FUNCTION_BLOCK "GCS7_E_MYFC_MOZF"	// FB 34
TITLE = MYFC/MOZF Liquids Flow Control
//  
//COPYRIGHT:    (C) 2002  BUHLER AG, CH-9240 UZWIL, SWITZERLAND
//
//PRODUCT:      GCS7
//
//TITLE:        Element MYFC/MOZF Liquids Flow Control
//
//-------------------------------------------------------------------------
//
//IDENT:        AUTHOR:             DEPT:                      DATE:
//
//FB34.3.1      A.Egli              CT3                        01-Dec-2005
//              Parameter Upload Change DBD86-->DBD88
//FB34.3.0      A.Egli              CT3                        05-Jan-2005
//              Parameter Upload (uses DB10)
//FB34.2.3      S.Cable             CDDP                       22-Mar-2004
//              Replace T D [AR1,xxx] with T LD [AR1,xxx]
//              If in Local, but released locally, do not alarm
//FB34.2.2      K.Tischer           CT3                        14-Jan-2004
//              Handling von InManual 
//FB34.2.1      A.Egli              CT3                        22-Dec-2003
//              StCode=6 also when StWaiting                
//FB34.2.0      A.Egli              CT3                        11-Dec-2003
//              InRestdischarge, StCode=6=Emptying 16=Emptying.Warning
//FB34.1.1      A.Egli              CT3                        17-Nov-2003
//              Alarm 90: Fault not DPRemoteControl
//FB34.1.0      A. Egli             CT3                        02-Jun-2002
//              1st Release in S7
//
//-------------------------------------------------------------------------
//
//PURPOSE:      MANUAL : see [MYFCxxMAN]
//
//RESTRICTIONS: S7
//-------------------------------------------------------------------------
//
//=======================================================
//Log Message: 
//------------------------------------------------------
//0     = Fault Cannceled
//1..79 = AlarmLC : Alarmnumber see manual of MYFC
//90   = Remote Control
//91   = StStopped
//92   = StDosing
//93   = StWaiting
//94   = Timeout starting
//95   = Timeout stopping
//96   = Communication fault
//97   = FaultManualMode
//98   = FaultLocalMode
//
//=======================================================
//StCode:  State               
//------------------------------------------------------
//32  StFault         
// 1  StStoppped      
// 2  StStarting      
// 3  StDosing        
//13  StDosing.Manual  
// 4  StWaiting       
// 7  StStopping      
//41  Stopped.HWStop        = StStopped + InHWStop
//51  Stopped.DPFault       = StStopped + InDPFault
//
AUTHOR : EA
FAMILY : GCS7LL
NAME : MYFCMOZE
VERSION : 3.1
VAR
  StCode : INT ;	//Element state code
  InEnable : BOOL ;	//Enable to dosing water
  InLocalWaterControl : BOOL ;	//1=Local Water Control enabled
  InManualWaterControl : BOOL ;	//1=Manual controled water enabled
  InSimulation : BOOL ;	//Simulation with DPSim (only DP)
  InRestdischarge : BOOL ;
  CmdNewJob : BOOL ;	//Clear actual values
  InHWStop : BOOL ;	//No Fault, Element changes to StStopped
  InDPFault : BOOL ;	//No Fault, Element changes to StStopped
  CmdOff : BOOL ;	//Pulse to stopp the element immediately (manual mode)
  CmdOn : BOOL ;	//Pulse to start  the element immediately (manual mode)
  CmdNext : BOOL ;	//Pulse to start the element in automatic mode (see global flags)
  CmdFaultReset : BOOL ;	//Command to reset fault
  InLocal : BOOL ;	//1= Local mode (no fault by start with service switch)
  InManual : BOOL ;	//1=Manual/ 0=Automatic
  InReport : BOOL ;	//Report of all state transitions
  spare37 : BOOL ;
  OutFaultCom : BOOL ;	//Communication fault
  OutFaultMode : BOOL ;	//Wrong mode
  OutFaultRelevant : BOOL ;	//Relevant fault MYFC or MOZF
  spare0403 : BOOL ;
  spare0404 : BOOL ;
  spare0405 : BOOL ;
  OutpEnable : BOOL ;	//24 V Enable signal water dosing
  OutWrongValue : BOOL ;	//Wrong nominal values, rejected by MEAF
  StStopped : BOOL ;	//Element is disabled
  StStarting : BOOL ;	//Element is starting
  StStopping : BOOL ;	//Element is sopping
  StDosing : BOOL ;	//Element is dosing
  StFault : BOOL ;	//Element has a communication or device fault
  StWaiting : BOOL ;	//Element is enabled, Waiting for Product
  OutWarning : BOOL ;	//Warning
  InMoisture : DINT ;	//[0.0 ... 99.9%] or [0..6500.0 l/h]     Is send to LC
  InOffsetMoisture : INT ;	//[-99.99 ... 99.99%]    Is send to MYFC
  InDosingMax : DINT ;	//[0.0 .. 99999.9 l/h] Is send to MYFC
  InProductGroup : INT ;	//[0..99]              Is send to MYFC
  spare18 : DINT ;
  OutMoisture : INT ;	//[0.0 ... 99.9%]      Is read from LC
  OutFlowrateProduct : DINT ;	//[0.. 999999 kg/h]    Is read from MYFC  [de: Istleistung Produkt]
  OutFlowrateWater : DINT ;	//[0.. 6500.0 l/h]    Is read from LC  [de: Istleistung MOZF]
  OutAlarmNrMYFC : INT ;	//Is read from MYFC
  OutAlarmNrMOZF : INT ;	//Is read from LC
  OutTotalProduct : DINT ;	//Is calculated by element
  OutTotalWater : DINT ;	//Is calculated by element
  OutNotErasableWater : DINT ;	//[0..99'999'999.9 l]  Is read from LC
  OutNotErasableProduct : DINT ;	//[0..999'999'999 kg]  Is read from MYFC
  spare52 : DINT ;
  spare56 : INT ;
  OutAlarmNrLog : INT ;
  Par : STRUCT
   ParObjectNo : INT ;	//Is used for communication with PC, e.g. for message
   ParMsgType : INT ;	//Is used for message (translation of state)
   ParHornCode : INT ;	//Is used by horn module
   ParLogOff : BOOL ;	//Report is off
   ParManual : BOOL ;	//Manual mode without interlocking
   ParMOZF : BOOL ;	//1=MOZF / 0=MYFC
   ParDP : BOOL ;	//1=DP / 0=Opto22
   ParFilter : STRUCT
    A05_24VToLow : BOOL ;
    A07ADRange : BOOL ;
    A08ADCalibration : BOOL ;
    A09ADFunction : BOOL ;
    A10ADSupply : BOOL ;
    A11AnalogInput : BOOL ;
    AxxCommunication : BOOL ;	//A12: Serial Interface ; A14=DPFault
    A17InternalCom : BOOL ;
    A26Tolerance : BOOL ;
    A30ZeroTara : BOOL ;
    A38Slide : BOOL ;
    A39Leck : BOOL ;
    A54RelaisMOZF : BOOL ;
    A55Moisture : BOOL ;
    A56TemperatureInternal : BOOL ;
    A57TemperatureExternal : BOOL ;
    A58SignalDumping : BOOL ;
    A59BulkDesity : BOOL ;
    A60Niveau : BOOL ;
    A63LevelProbe : BOOL ;
    A64AlarmMOZE : BOOL ;
    A65MinFlowrate : BOOL ;
    A66MaxFlowrate : BOOL ;
    A67ToleranceWater : BOOL ;
   END_STRUCT ;
   ParComDB : INT ;	//OPTO22: Communication DB
   ParLCIdx : INT ;	//OPTO22: Index of data record
   ParLCAddr : INT ;	//OPTO22: Address of LC Opto22
   ParIOByteNr : INT ;	//PROFIBUS: Address of first input and output byte
   ParMonTime : INT  := 20;	//After this time outputs must be equal inputs
   spare20 : DINT ;
   spare24 : DINT ;
   OutMonTime : INT ;	//Actual time: Monitoring
   OutFlags : STRUCT
    OutFaultResetDone : BOOL ;
    OutAlarmReadAgain : BOOL ;
    OutTestNewAlarm : BOOL ;
    OutRelevantFaultMOZF : BOOL ;	//Relevant fault number
    OutRelevantFaultMYFC : BOOL ;	//Relevant fault number
    OutNoAlarmMOZF : BOOL ;	//Alarmnumber 0 is read form LC
    OutNoAlarmMYFC : BOOL ;	//Alarmnumber 0 is read form LC
    OutComFaultRead : BOOL ;	//Only DP
    OutComFaultSend : BOOL ;	//Only DP
    spare03 : BOOL ;
    spare04 : BOOL ;
    spare05 : BOOL ;
   END_STRUCT ;
   Command : STRUCT 	//Only used with DP Communication
    spare10 : BOOL ;
    spare11 : BOOL ;
    InRestdischarge : BOOL ;
    spare13 : BOOL ;
    spare14 : BOOL ;
    spare15 : BOOL ;
    spare16 : BOOL ;
    AcceptNewDataReady : BOOL ;	//de: Quittierung neue Werte Bereit
    spare2 : BYTE ;
    spare3 : BYTE ;
    CommandReady : BOOL ;	//de: Steuersignale gültig
    spare41 : BOOL ;
    spare42 : BOOL ;
    spare43 : BOOL ;
    spare44 : BOOL ;
    ResetAlarm : BOOL ;	//de: Alarm löschen
    NewSendData : BOOL ;	//de: Aenderung Sendedaten
    AcceptNewRcvData : BOOL ;	//de: Quittierung Aenderung Empfangsdatensatz
   END_STRUCT ;
   Status : STRUCT 	//Only used with DP Communication
    Enable24V : BOOL ;	//Dosing release
    Dosing : BOOL ;	//de: Wasser dosiert
    Remote : BOOL ;	//Remote=1 /Local=0
    Manual : BOOL ;	//de: Hand
    Level : BOOL ;	//1=Covered  de: Sonde Netzgeraet
    Active : BOOL ;	//de: Netzung aktiv
    spare16 : BOOL ;
    NewDataReady : BOOL ;	//de: Neue Werte Bereit
    spare2 : BYTE ;
    spare3 : BYTE ;
    spare40 : BOOL ;
    spare41 : BOOL ;
    spare42 : BOOL ;	//de: Stuerung Remote
    RemoteControlDP : BOOL ;	//de: Sollwertvorgabe Remote
    WrongValue : BOOL ;	//de: Falscher Sollwert
    SumFault : BOOL ;	//de: Sammelalarm
    AcceptNewSendData : BOOL ;	//de: Quittierung Aenderung Sendedaten
    NewRcvData : BOOL ;	//de: Aenderung Empfangsdaten
   END_STRUCT ;
  END_STRUCT ;
END_VAR
VAR_TEMP
  tmpFilter : ARRAY  [0 .. 95 ] OF BOOL ;
  tmpLOGvalue : WORD ;	//LOG value
  tmpCommand : INT ;
  tmpFBNO : INT ;	//Number of the actual FB
  tmpFault : BOOL ;
  tmpOff : BOOL ;
  tmpOn : BOOL ;
  tmpLocal : BOOL ;
  tmpEnable : BOOL ;
  tmpReport : BOOL ;
  tmpLenDyn : DINT ;
  tmpAddr : WORD ;
  tmpReturn : INT ;
  tmpComDB : INT ;
  Set001 : STRUCT
   OutMoistureAc : BYTE ;	//[0.0 ... 99.9%]      Is read from LC
   spare9 : BYTE ;
   OutFlowRateMOZF : INT ;	//[0.. 99999.9 l/h]    Is read from LC  [de: Istleistung MOZF]
   OutFlowRateProduct : DINT ;	//[0.. 999999 kg/h]    Is read from MYFC  [de: Istleistung Produkt]
   OutNotErasableTotalWater : DINT ;	//[0..99'999'999.9 l]  Is read from LC
   spare20 : BYTE ;
   OutRecipeNr : BYTE ;
   OutAlarmNumberMYFC : BYTE ;	//Is read from MYFC
   OutAlarmNumberMOZF : BYTE ;	//Is read from LC
  END_STRUCT ;
  Set136 : STRUCT
   InMoistureNom : INT ;	//[0.00 ... 25.0%]      Is send to LC
   spare10 : INT ;
   InMoistureOffset : INT ;	//[-99.99 ... 99.99%]    Is send to MYFC
   InDosingMax : WORD ;	//[0.0 .. 99999.9 l/h] Is send to MYFC
   InProductGroup : BYTE ;	//[0..99]              Is send to MYFC
   Spare17 : BYTE ;
   Spare18 : DWORD ;
   Spare22 : WORD ;
  END_STRUCT ;
  DPData : STRUCT
   StatusCommand : DWORD ;
   NrSndDataSet : BYTE ;	//de: Nummer Sendedatensatz
   IdxSndDataSet : BYTE ;	//de: Index Sendedatensatz
   NrRcvDataSet : BYTE ;	//de: Nummer Empfangsdatensatz
   IdxRcvDataSet : BYTE ;	//de: Index Empfangsdatensatz
   Data : ARRAY  [1 .. 4 ] OF DINT ;
  END_STRUCT ;
  tmpWtWater : DINT ;
  tmpWtProduct : DINT ;
  tmpCalculate : BOOL ;
  tmpNewAlarmNumber : BOOL ;
  tmpCallBackFuction : BOOL ;	//Call back function is active
  tmpFaultMonitoringStart : BOOL ;
  tmpFaultMonitoringStop : BOOL ;
END_VAR
BEGIN
NETWORK
TITLE =  Start Global
      L     #Par.ParComDB;
      T     #tmpComDB;
      L     34;
      T     #tmpFBNO;
      L     102;
      T     #tmpLenDyn;	//--> Len dynamic data in byte
      SET;
      R     #tmpCalculate;
      R     #tmpCallBackFuction;
      R     #tmpNewAlarmNumber;
      R     #tmpFaultMonitoringStart;
      R     #tmpFaultMonitoringStop;
//tmpLocal
      A     #InLocal;
      AN    #InManual;
      =     #tmpLocal;
NETWORK
TITLE =
      LAR1  P##tmpFilter;
      L     0;
      T     LD [AR1,P#0.0];	//tmpFilter[00..31] [2.3]
      T     LD [AR1,P#0.0];	//tmpFilter[32..63] [2.3]
      T     LD [AR1,P#0.0];	//tmpFilter[64..95] [2.3]
      SET;
      S     #tmpFilter[13];
      S     #tmpFilter[18];
      A     #Par.ParFilter.A05_24VToLow;
      =     #tmpFilter[5];
      A     #Par.ParFilter.A07ADRange;
      =     #tmpFilter[7];
      A     #Par.ParFilter.A08ADCalibration;
      =     #tmpFilter[8];
      A     #Par.ParFilter.A09ADFunction;
      =     #tmpFilter[9];
      A     #Par.ParFilter.A10ADSupply;
      =     #tmpFilter[10];
      A     #Par.ParFilter.A11AnalogInput;
      =     #tmpFilter[11];
      A     #Par.ParFilter.AxxCommunication;
      =     #tmpFilter[12];
      =     #tmpFilter[14];
      A     #Par.ParFilter.A17InternalCom;
      =     #tmpFilter[17];
      A     #Par.ParFilter.A26Tolerance;
      =     #tmpFilter[26];
      A     #Par.ParFilter.A30ZeroTara;
      =     #tmpFilter[30];
      A     #Par.ParFilter.A38Slide;
      =     #tmpFilter[38];
      A     #Par.ParFilter.A39Leck;
      =     #tmpFilter[39];
      A     #Par.ParFilter.A54RelaisMOZF;
      =     #tmpFilter[54];
      A     #Par.ParFilter.A55Moisture;
      =     #tmpFilter[55];
      A     #Par.ParFilter.A56TemperatureInternal;
      =     #tmpFilter[56];
      A     #Par.ParFilter.A57TemperatureExternal;
      =     #tmpFilter[57];
      A     #Par.ParFilter.A58SignalDumping;
      =     #tmpFilter[58];
      A     #Par.ParFilter.A59BulkDesity;
      =     #tmpFilter[59];
      A     #Par.ParFilter.A60Niveau;
      =     #tmpFilter[60];
      A     #Par.ParFilter.A63LevelProbe;
      =     #tmpFilter[63];
      A     #Par.ParFilter.A64AlarmMOZE;
      =     #tmpFilter[64];
      A     #Par.ParFilter.A65MinFlowrate;
      =     #tmpFilter[65];
      A     #Par.ParFilter.A66MaxFlowrate;
      =     #tmpFilter[66];
      A     #Par.ParFilter.A67ToleranceWater;
      =     #tmpFilter[67];
NETWORK
TITLE =  Call back function (***Opto22***)
////*************************************************
////***             O P T O 22                    ***
////*************************************************
//
//This functions are called by FBxxx (COM) 
      A     #Par.ParDP;
      JC    PC;
      OPN   DB [#tmpComDB];
      L     0;
      L     DBW 32;	//COM.Element.CODE;
      ==I;
      JC    PC;
//Check if object has moved
      L     #Par.ParObjectNo;
      L     DBD 60;	//COM.LC0.AddrPara;       
      ==D;
      JC    COok;
      BEC;
//=============================================
COok: S     #tmpCallBackFuction;
      L     DBB 76;	//COM.Telegram.Command;
      T     #tmpCommand;
      L     1;
      L     DBW 32;	//COM.Element.CODE;
      ==I;
      JC    Send;
      L     2;
      ==I;
      JC    Rcv;
      L     4;	//NAK
      L     DBW 32;	//COM.Element.CODE;
      ==I;
      S     #OutFaultCom;	//fault MYEB communication
      BEU;
//--------------------------
//Send C
//--------------------------
Send: NOP   0;
      L     #tmpCommand;
      L     'C';
      <>I;
      JC    SndF;
// command 1
      A     #CmdFaultReset;
      =     #Par.Command.ResetAlarm;
      R     #CmdFaultReset;
// command 1
      L     0;	//Character offset
      T     DBW 40;	//COM.Element.AddrOffset
      L     0;
      T     DBD 36;	//COM.Element.InOutValue
      A     #Par.Command.ResetAlarm;
      =     DBX 39.0;	//-->ResetAlarm
      A     #InRestdischarge;	//                        [2.0]
      =     DBX 39.1;	//-->InRestdischarge      [2.0]
      A     #OutpEnable;
      =     DBX 39.7;	//-->Enable24V for OPTOSIM
      L     32;	//Convert Hex to 2-ASCII
      T     DBW 0;	//COM.CODE
      CDB;	//ComDB->Instanz-DB
      UC    "GCS7_RS485Ctrl";	//Convert (CODE=DBW0)
      CDB;	//ElementDB->Instanz-DB
// InMoistureNom    
      L     2;	//Character offset
      T     DBW 40;	//COM.Element.AddrOffset
      L     #InMoisture;
      T     DBD 36;	//COM.Element.InOutValue
      L     13;	//Convert DInt to 3-ASCII
      T     DBW 0;	//COM.CODE
      CDB;	//ComDB->Instanz-DB
      UC    "GCS7_RS485Ctrl";	//Convert (CODE=DBW0)
      CDB;	//ElementDB->Instanz-DB
// InMoistureOffset    
      L     5;	//Character offset
      T     DBW 40;	//COM.Element.AddrOffset
      L     #InOffsetMoisture;	//[4.0]
      T     DBD 36;	//COM.Element.InOutValue
      L     15;	//Convert DInt to 5-ASCII
      T     DBW 0;	//COM.CODE
      CDB;	//ComDB->Instanz-DB
      UC    "GCS7_RS485Ctrl";	//Convert (CODE=DBW0)
      CDB;	//ElementDB->Instanz-DB
// InDosingMax    
      L     10;	//Character offset
      T     DBW 40;	//COM.Element.AddrOffset
      L     #InDosingMax;	// 
      T     DBD 36;	//COM.Element.InOutValue
      L     16;	//Convert DInt to 6-ASCII
      T     DBW 0;	//COM.CODE
      CDB;	//ComDB->Instanz-DB
      UC    "GCS7_RS485Ctrl";	//Convert (CODE=DBW0)
      CDB;	//ElementDB->Instanz-DB
// InProductGroup    
      L     16;	//Character offset
      T     DBW 40;	//COM.Element.AddrOffset
      L     #InProductGroup;	// 
      T     DBD 36;	//COM.Element.InOutValue
      L     12;	//Convert DInt to 2-ASCII
      T     DBW 0;	//COM.CODE
      CDB;	//ComDB->Instanz-DB
      UC    "GCS7_RS485Ctrl";	//Convert (CODE=DBW0)
      CDB;	//ElementDB->Instanz-DB
// spare    
      L     18;	//Character offset
      T     DBW 40;	//COM.Element.AddrOffset
      L     0;	// 
      T     DBD 36;	//COM.Element.InOutValue
      L     18;	//Convert DInt to 8-ASCII
      T     DBW 0;	//COM.CODE
      CDB;	//ComDB->Instanz-DB
      UC    "GCS7_RS485Ctrl";	//Convert (CODE=DBW0)
      CDB;	//ElementDB->Instanz-DB
// spare    
      L     24;	//Character offset
      T     DBW 40;	//COM.Element.AddrOffset
      L     0;	// 
      T     DBD 36;	//COM.Element.InOutValue
      L     16;	//Convert DInt to 6-ASCII
      T     DBW 0;	//COM.CODE
      CDB;	//ComDB->Instanz-DB
      UC    "GCS7_RS485Ctrl";	//Convert (CODE=DBW0)
      CDB;	//ElementDB->Instanz-DB
      L     30;	//Lenght in byte
      T     DBW 78;	//COM.Telegram.Len
      L     50;	//Lenght in byte
      T     DBW 86;	//COM.Telegram.LenAnswer
      BEU;
//--------------------------
//Send F
//--------------------------
SndF: NOP   0;
      L     #tmpCommand;
      L     'F';
      <>I;
      JC    SndZ;
// command 1
      A     #CmdFaultReset;
      =     #Par.Command.ResetAlarm;
      R     #CmdFaultReset;
// command 1
      L     0;	//Character offset
      T     DBW 40;	//COM.Element.AddrOffset
      L     0;
      T     DBD 36;	//COM.Element.InOutValue
      A     #Par.Command.ResetAlarm;
      =     DBX 39.0;	//-->ResetAlarm
      A     #OutpEnable;
      =     DBX 39.7;	//-->Enable24V for OPTOSIM
      L     32;	//Convert Hex to 2-ASCII
      T     DBW 0;	//COM.CODE
      CDB;	//ComDB->Instanz-DB
      UC    "GCS7_RS485Ctrl";	//Convert (CODE=DBW0)
      CDB;	//ElementDB->Instanz-DB
// InMoistureNom    
      L     2;	//Character offset
      T     DBW 40;	//COM.Element.AddrOffset
      L     #InMoisture;
      T     DBD 36;	//COM.Element.InOutValue
      L     16;	//Convert DInt to 6-ASCII
      T     DBW 0;	//COM.CODE
      CDB;	//ComDB->Instanz-DB
      UC    "GCS7_RS485Ctrl";	//Convert (CODE=DBW0)
      CDB;	//ElementDB->Instanz-DB
// spare    
      L     8;	//Character offset
      T     DBW 40;	//COM.Element.AddrOffset
      L     0;	// 
      T     DBD 36;	//COM.Element.InOutValue
      L     12;	//Convert DInt to 2-ASCII
      T     DBW 0;	//COM.CODE
      CDB;	//ComDB->Instanz-DB
      UC    "GCS7_RS485Ctrl";	//Convert (CODE=DBW0)
      CDB;	//ElementDB->Instanz-DB
      L     10;	//Lenght in byte
      T     DBW 78;	//COM.Telegram.Len
      L     30;	//Lenght in byte
      T     DBW 86;	//COM.Telegram.LenAnswer
SndZ: BEU;
//--- Get done ---------------
//Copy reveived data to element
//--------------------------
//Receive C
//--------------------------
Rcv:  R     #OutFaultCom;
      L     #tmpCommand;
      L     'C';
      <>I;
      JC    RcvF;
      A     #Par.OutFlags.OutFaultResetDone;	//[1.2]
      S     #Par.OutFlags.OutTestNewAlarm;	//[1.2]
      A     #Par.Command.ResetAlarm;	//    [1.2]
      =     #Par.OutFlags.OutFaultResetDone;	// [1.2] 
//LC status
      L     0;	//Character offset
      T     DBW 40;	//COM.Element.AddrOffset
      L     42;	//Convert 2-ASCII to Hex
      T     DBW 0;	//COM.CODE
      CDB;	//ComDB->Instanz-DB
      UC    "GCS7_RS485Ctrl";	//Convert (CODE=DBW0)
      CDB;	//ElementDB->Instanz-DB
      CALL  "SIEMENS_BLKMOV" (
           SRCBLK                   := DBB 39,
           RET_VAL                  := #tmpReturn,
           DSTBLK                   := #Par.Status);
//OutMoistureAc
      L     2;	//Character offset
      T     DBW 40;	//COM.Element.AddrOffset
      L     23;	//Convert 3-ASCII to DInt
      T     DBW 0;	//COM.CODE
      CDB;	//ComDB->Instanz-DB
      UC    "GCS7_RS485Ctrl";	//Convert (CODE=DBW0)
      CDB;	//ElementDB->Instanz-DB
      L     DBD 36;	//COM.Element.InOutValue
      T     #OutMoisture;
//OutFlowRateProduct
      L     5;	//Character offset
      T     DBW 40;	//COM.Element.AddrOffset
      L     26;	//Convert 6-ASCII to DInt
      T     DBW 0;	//COM.CODE
      CDB;	//ComDB->Instanz-DB
      UC    "GCS7_RS485Ctrl";	//Convert (CODE=DBW0)
      CDB;	//ElementDB->Instanz-DB
      L     DBD 36;	//COM.Element.InOutValue
      T     #OutFlowrateProduct;
//OutFlowRateMOZF
      L     11;	//Character offset
      T     DBW 40;	//COM.Element.AddrOffset
      L     26;	//Convert 6-ASCII to DInt
      T     DBW 0;	//COM.CODE
      CDB;	//ComDB->Instanz-DB
      UC    "GCS7_RS485Ctrl";	//Convert (CODE=DBW0)
      CDB;	//ElementDB->Instanz-DB
      L     DBD 36;	//COM.Element.InOutValue
      T     #OutFlowrateWater;
//OutNotErasableTotalWater
      L     17;	//Character offset
      T     DBW 40;	//COM.Element.AddrOffset
      L     29;	//Convert 9-ASCII to DInt
      T     DBW 0;	//COM.CODE
      CDB;	//ComDB->Instanz-DB
      UC    "GCS7_RS485Ctrl";	//Convert (CODE=DBW0)
      CDB;	//ElementDB->Instanz-DB
      L     DBD 36;	//COM.Element.InOutValue
      T     #tmpWtWater;
//OutNotErasableTotalProd
      L     26;	//Character offset
      T     DBW 40;	//COM.Element.AddrOffset
      L     29;	//Convert 9-ASCII to DInt
      T     DBW 0;	//COM.CODE
      CDB;	//ComDB->Instanz-DB
      UC    "GCS7_RS485Ctrl";	//Convert (CODE=DBW0)
      CDB;	//ElementDB->Instanz-DB
      L     DBD 36;	//COM.Element.InOutValue
      T     #tmpWtProduct;
//OutAlarmNumberMYFC
      L     35;	//Character offset
      T     DBW 40;	//COM.Element.AddrOffset
      L     22;	//Convert 2-ASCII to DInt
      T     DBW 0;	//COM.CODE
      CDB;	//ComDB->Instanz-DB
      UC    "GCS7_RS485Ctrl";	//Convert (CODE=DBW0)
      CDB;	//ElementDB->Instanz-DB
      L     DBD 36;	//COM.Element.InOutValue
      T     #Set001.OutAlarmNumberMYFC;
//OutAlarmNumberMOZF
      L     37;	//Character offset
      T     DBW 40;	//COM.Element.AddrOffset
      L     22;	//Convert 2-ASCII to DInt
      T     DBW 0;	//COM.CODE
      CDB;	//ComDB->Instanz-DB
      UC    "GCS7_RS485Ctrl";	//Convert (CODE=DBW0)
      CDB;	//ElementDB->Instanz-DB
      L     DBD 36;	//COM.Element.InOutValue
      T     #Set001.OutAlarmNumberMOZF;
      SET;
      S     #tmpCalculate;
      S     #tmpNewAlarmNumber;
      JU    RCal;	// -->Calculate
//--------------------------
//Receive F
//--------------------------
RcvF: R     #OutFaultCom;
      L     #tmpCommand;
      L     'F';
      <>I;
      BEC;
      A     #Par.OutFlags.OutFaultResetDone;	//[1.2]
      S     #Par.OutFlags.OutTestNewAlarm;	//[1.2]
      A     #Par.Command.ResetAlarm;	//    [1.2]
      R     #CmdFaultReset;
      =     #Par.OutFlags.OutFaultResetDone;	// [1.2] 
//LC status
      L     0;	//Character offset
      T     DBW 40;	//COM.Element.AddrOffset
      L     42;	//Convert 2-ASCII to Hex
      T     DBW 0;	//COM.CODE
      CDB;	//ComDB->Instanz-DB
      UC    "GCS7_RS485Ctrl";	//Convert (CODE=DBW0)
      CDB;	//ElementDB->Instanz-DB
      L     DBD 36;	//COM.Element.InOutValue
      CALL  "SIEMENS_BLKMOV" (
           SRCBLK                   := DBB 39,
           RET_VAL                  := #tmpReturn,
           DSTBLK                   := #Par.Status);
//OutFlowRateMOZF
      L     2;	//Character offset
      T     DBW 40;	//COM.Element.AddrOffset
      L     26;	//Convert 6-ASCII to DInt
      T     DBW 0;	//COM.CODE
      CDB;	//ComDB->Instanz-DB
      UC    "GCS7_RS485Ctrl";	//Convert (CODE=DBW0)
      CDB;	//ElementDB->Instanz-DB
      L     DBD 36;	//COM.Element.InOutValue
      T     #OutFlowrateWater;
//OutNotErasableTotalWater
      L     8;	//Character offset
      T     DBW 40;	//COM.Element.AddrOffset
      L     29;	//Convert 9-ASCII to DInt
      T     DBW 0;	//COM.CODE
      CDB;	//ComDB->Instanz-DB
      UC    "GCS7_RS485Ctrl";	//Convert (CODE=DBW0)
      CDB;	//ElementDB->Instanz-DB
      L     DBD 36;	//COM.Element.InOutValue
      T     #tmpWtWater;
      L     0;
      T     #tmpWtProduct;
//OutAlarmNumberMOZF
      L     17;	//Character offset
      T     DBW 40;	//COM.Element.AddrOffset
      L     22;	//Convert 2-ASCII to DInt
      T     DBW 0;	//COM.CODE
      CDB;	//ComDB->Instanz-DB
      UC    "GCS7_RS485Ctrl";	//Convert (CODE=DBW0)
      CDB;	//ElementDB->Instanz-DB
      L     DBD 36;	//COM.Element.InOutValue
      T     #Set001.OutAlarmNumberMOZF;
      L     0;
      T     #Set001.OutAlarmNumberMYFC;
      SET;
      S     #tmpCalculate;
      S     #tmpNewAlarmNumber;
      JU    RCal;	//-->Calculate Total
NETWORK
TITLE = PC Control
//=== Test Object number =====================
PC:   L     "SYS_DirectCtrlDB".PC.ObjectNo;	//PCControl.ObjectNo
      L     #Par.ParObjectNo;	//Input ObjectNo
      <>I;
      JC    Ctrl;
//=== Test OType      ========================
      L     1034;	//Input object type
      L     "SYS_DirectCtrlDB".PC.ObjectType;	//PCControl.ObjectType
      <>I;
      JC    Ctrl;
//=== Test Handshake =========================
      A     "SYS_DirectCtrlDB".PC.Hsk.FExamine;	//Handshake.FExamine
      JC    pExa;
      A     "SYS_DirectCtrlDB".PC.Hsk.FDefineCmd;	//Handshake.FDefineCmd
      JC    pCmd;
      A     "SYS_DirectCtrlDB".PC.Hsk.FDefinePara;	//Handshake.FDefinePara
      JC    pPar;
pIni: L     2;	//FcInit
      UC    "SYS_DirectCtrl";
      JU    Ctrl;
// Write parameter 
pPar: LAR1  P#DBX 58.0;	//PCControl.Value[1]
      L     #tmpLenDyn;
      SLD   3;
      +AR1;	//PCControl.Value[x]
      L     DBW [AR1,P#20.0];	//PCControl.Value[x+6]
      T     #Par.ParMonTime;
//Write new commands from PC to Interface of group 
pCmd: A     "SYS_DirectCtrlDB".PC.Cmd1[8];	// CmdOff
      AN    "GCS7_Gr_OutManualOff";	//Global.OutManualOff 
      S     #CmdOff;
      A     "SYS_DirectCtrlDB".PC.Cmd1[9];	// CmdOn
      AN    "GCS7_Gr_OutManualOff";	//Global.OutManualOff
      S     #CmdOn;
      A     "SYS_DirectCtrlDB".PC.Cmd1[10];	// CmdNext
      S     #CmdNext;
      A     "SYS_DirectCtrlDB".PC.Cmd1[11];	// CmdFaultReset
      S     #CmdFaultReset;
      A     "SYS_DirectCtrlDB".PC.Cmd1[1];	//Cmd1[1]
      S     #InLocalWaterControl;
      R     #InManualWaterControl;	// CmdManualOn
      A     "SYS_DirectCtrlDB".PC.Cmd1[2];
      S     #InManualWaterControl;	// CmdReportOn
      A     "SYS_DirectCtrlDB".PC.Cmd1[3];
      R     #InLocalWaterControl;	// CmdManualOff
      R     #InManualWaterControl;
      A     "SYS_DirectCtrlDB".PC.Cmd1[5];	//Cmd1[5]  =CmdNewJob
      S     #CmdNewJob;
      A     "SYS_DirectCtrlDB".PC.Cmd1[13];	// CmdManualOn
      S     #InManual;
      A     "SYS_DirectCtrlDB".PC.Cmd1[14];	// CmdReportOn
      S     #InReport;
      A     "SYS_DirectCtrlDB".PC.Cmd2[13];	// CmdManualOff
      R     #InManual;
      A     "SYS_DirectCtrlDB".PC.Cmd2[14];	// CmdReportOff
      R     #InReport;
//Define Value
      AN    "SYS_DirectCtrlDB".PC.Hsk.FDefineValue;	// PC.Hsk.FDefineValue
      ON    #InManual;
      JC    pIni;
      LAR1  P#DBX 58.0;
      L     DBD [AR1,P#6.0];
      T     #InMoisture;
      L     DBW [AR1,P#10.0];
      T     #InOffsetMoisture;
      L     DBD [AR1,P#12.0];
      T     #InDosingMax;
      L     DBW [AR1,P#16.0];
      T     #InProductGroup;
      JU    pIni;
pExa: TAR2;	//Address dynamic datas
      T     "SYS_DirectCtrlDB".GC.InDynAddr;	//-->PCControl.GC.InDynAddr
      L     #tmpLenDyn;	//Length dynamic datas
      T     "SYS_DirectCtrlDB".GC.InDynLen;	//-->PCControl.GC.InDynLen
      L     0;	//Address parameter data
      T     "SYS_DirectCtrlDB".GC.InParaAddr;	//-->PCControl.GC.InParaAddr
      L     0;	//Length parameter
      T     "SYS_DirectCtrlDB".GC.InParaLen;	//-->PCControl.GC.InParaLen
      L     1;	//Code FcExamine
      UC    "SYS_DirectCtrl";
      L     0;	//Revision
      T     "SYS_DirectCtrlDB".GC.Revision;
Ctrl: NOP   0;
NETWORK
TITLE = [3.0] LCParameter
      L     #Par.ParObjectNo;
      L     "SYS_DirectCtrlLCDB".PC.ObjectNo;
      <>I;
      O     #Par.ParDP;
      JC    LCP0;
      T     "SYS_DirectCtrlLCDB".GC.InObjectNo;
      L     #Par.ParComDB;
      T     "SYS_DirectCtrlLCDB".GC.InDBNr;
      L     #Par.ParLCAddr;
      T     "SYS_DirectCtrlLCDB".GC.InLCAddr;
LCP0: NOP   0;
NETWORK
TITLE = Read data from LC (**DP**)
////*************************************************
////***            DP Communication              ***
////*************************************************
//
      AN    #Par.ParDP;
      JC    rcv0;
      L     #Par.ParIOByteNr;
      T     #tmpAddr;
      A     #InSimulation;
      JC    rSim;
      CALL  "SIEMENS_DPRD_DAT" (
           LADDR                    := #tmpAddr,
           RET_VAL                  := #tmpReturn,
           RECORD                   := #DPData);
      L     #tmpReturn;
      L     0;
      <>I;
      =     #Par.OutFlags.OutComFaultRead;
      JC    rcv0;
      JU    rDP;
//read from Simulation
rSim: R     #Par.OutFlags.OutComFaultRead;
      A     "GCS7_Gr_SimDPtoImage";
      L     P#I 0.0;
      JC    rDB1;
      OPN   "TEST_IOSimuliInput";
      L     P#DBX 0.0;
rDB1: L     #Par.ParIOByteNr;
      SLD   3;
      +D;
      LAR1;
      L     D [AR1,P#0.0];
      T     #DPData.StatusCommand;
      L     B [AR1,P#4.0];
      T     #DPData.NrSndDataSet;
      L     B [AR1,P#5.0];
      T     #DPData.IdxSndDataSet;
      L     B [AR1,P#6.0];
      T     #DPData.NrRcvDataSet;
      L     B [AR1,P#7.0];
      T     #DPData.IdxRcvDataSet;
      L     D [AR1,P#8.0];
      T     #DPData.Data[1];
      L     D [AR1,P#12.0];
      T     #DPData.Data[2];
      L     D [AR1,P#16.0];
      T     #DPData.Data[3];
      L     D [AR1,P#20.0];
      T     #DPData.Data[4];
//==Copy Status===============
rDP:  L     #DPData.NrRcvDataSet;
      L     0;
      ==I;
      JC    R001;
      CALL  "SIEMENS_BLKMOV" (
           SRCBLK                   := #DPData.StatusCommand,
           RET_VAL                  := #tmpReturn,
           DSTBLK                   := #Par.Status);
      AN    #Par.Status.NewRcvData;
      A     #InSimulation;
      JC    rcv0;
//===============================
//Answer Dataset 001
      L     #DPData.NrRcvDataSet;
      L     1;
      <>I;
      JC    r11;	//[3.0]
      CALL  "SIEMENS_BLKMOV" (
           SRCBLK                   := #DPData.Data,
           RET_VAL                  := #tmpReturn,
           DSTBLK                   := #Set001);
      L     #Set001.OutMoistureAc;
      T     #OutMoisture;
      L     #Set001.OutFlowRateProduct;
      T     #OutFlowrateProduct;
      L     #Set001.OutFlowRateMOZF;
      T     #OutFlowrateWater;
//Reset old alarm flags with CmdFaultReset
      A     #Par.OutFlags.OutAlarmReadAgain;
      A     #Par.OutFlags.OutFaultResetDone;
      R     #Par.OutFlags.OutFaultResetDone;
      S     #Par.OutFlags.OutTestNewAlarm;
      A     #Par.OutFlags.OutFaultResetDone;
      =     #Par.OutFlags.OutAlarmReadAgain;
//--------------------------------------
//WtNotErasable
      L     #Set001.OutNotErasableTotalWater;
      T     #tmpWtWater;
      L     #OutNotErasableProduct;
      T     #tmpWtProduct;
// 
      SET;
      S     #tmpCalculate;	//--> Calculate job weight 
      S     #tmpNewAlarmNumber;	//--> Test new Alarm number
      JU    R11;	//[3.0]   
//===============================
//[7.0]--> LC Parameter 
//Reading dataset 11
R11:  L     "SYS_DirectCtrlLCDB".PC.ObjectNo;
      L     #Par.ParObjectNo;
      <>I;
      JC    R002;
      AN    "SYS_DirectCtrlLCDB".PC.Hsk.FExamineFirst;
      AN    "SYS_DirectCtrlLCDB".PC.Hsk.FExamineNext;
      JC    R002;
// -- Start Reading with Dataset 11
      L     11;
      T     #DPData.NrRcvDataSet;
      L     253;	//First
      A     "SYS_DirectCtrlLCDB".PC.Hsk.FExamineFirst;
      JC    rLC9;
      L     254;	//Next
rLC9: T     #DPData.IdxRcvDataSet;
      JU    rcv0;
//---Answer  dataset 11 ---
//---Answer  dataset 12 ---
r11:  L     #DPData.NrRcvDataSet;
      L     11;
      <>I;
      JC    rLCB;
// Answer Dataset 11
      L     '  ';
      T     "SYS_DirectCtrlLCDB".PC.Value[1];
      L     #DPData.Data[1];
      T     DB10.DBD 60;
      L     #DPData.Data[2];
      T     DB10.DBD 64;
      L     #DPData.Data[3];
      T     DB10.DBD 68;
      L     #DPData.Data[4];
      T     DB10.DBD 72;
      L     #DPData.IdxRcvDataSet;
      L     255;
      ==I;
      JC    rLCE;
      S     "SYS_DirectCtrlLCDB".GC.Set11Done;
      L     12;
      T     #DPData.NrRcvDataSet;
      L     0;
      T     #DPData.IdxRcvDataSet;
      JU    rcv0;	//--> Read dataset 12
// Answer Dataset 12
rLCB: L     #DPData.NrRcvDataSet;
      L     12;
      <>I;
      JC    r002;
      L     #DPData.Data[1];
      T     DB10.DBD 76;
      L     #DPData.Data[2];
      T     DB10.DBD 80;
      L     #DPData.Data[3];
      T     DB10.DBD 84;
      L     #DPData.Data[4];
      T     DB10.DBD 88;
      AN    "SYS_DirectCtrlLCDB".GC.Set11Done;
      JC    R002;
rLCE: L     12;
      CALL  "SYS_DirectCtrl";
      JU    R002;
//<--[3.0]
//===============================
//Answer  dataset 2
r002: L     #DPData.NrRcvDataSet;
      L     2;
      <>I;
      JC    R001;
      L     #DPData.Data[1];	//WtActual
      T     #tmpWtProduct;
      L     #OutNotErasableWater;
      T     #tmpWtWater;
      SET;
      S     #tmpCalculate;	//--> Calculate job weight 
      JU    R001;
//===============================
//Read Dataset 001
R001: L     1;
      T     #DPData.NrRcvDataSet;
      L     0;
      T     #DPData.IdxRcvDataSet;
      JU    rcv0;
//===============================
//Read Dataset 002
R002: A     #Par.ParMOZF;
      JC    R001;
      L     2;
      T     #DPData.NrRcvDataSet;
      L     0;
      T     #DPData.IdxRcvDataSet;
      JU    rcv0;
rcv0: NOP   0;
NETWORK
TITLE = Calculate total / store alarm number (DP and OPTO22)
      AN    #tmpCalculate;
      JC    rEnd;
//===================================
//Calculate total Water 
//===================================
//---  Init first, if old value < 0  
RCal: L     #OutNotErasableWater;
      L     0;
      <D;
      JC    rWZ2;
//---  Calculate Weight ---
      L     #tmpWtWater;
      L     #OutNotErasableWater;
      -D;
      JM    rWZ1;
      JU    rWPo;
rWZ1: L     L#1000000000;
      +D;
rWPo: L     10000;	// Maximum change by relaod software
      >D;
      JC    rWZ2;
      TAK;
      L     #OutTotalWater;
      +D;
      T     #OutTotalWater;
rWZ2: L     #tmpWtWater;
      T     #OutNotErasableWater;
//===================================
//Calculate total Prod 
//===================================
//---  Init first, if old value < 0  
      L     #OutNotErasableProduct;
      L     0;
      <D;
      JC    rPZ2;
//---  Calculate Weight ---
      L     #tmpWtProduct;
      L     #OutNotErasableProduct;
      -D;
      JM    rPZ1;
      JU    rPPo;
rPZ1: L     L#1000000000;
      +D;
rPPo: L     10000;	// Maximum change by relaod software
      >D;
      JC    rPZ2;
      TAK;
      L     #OutTotalProduct;
      +D;
      T     #OutTotalProduct;
rPZ2: L     #tmpWtProduct;
      T     #OutNotErasableProduct;
//===================================
//Store Alarmnumber
//===================================
      AN    #tmpNewAlarmNumber;	//--> Test new Alarm number
      JC    r000;
//--- keep old alalrm number  MOZF ----
      L     0;
      L     #Set001.OutAlarmNumberMOZF;
      ==I;
      =     #Par.OutFlags.OutNoAlarmMOZF;
//      U     #OutFlags.OutNoAlarmMOZF
      A     #Par.OutFlags.OutRelevantFaultMOZF;
      AN    #Par.OutFlags.OutTestNewAlarm;
      AN    #tmpLocal;
      AN    #InManual;
      JC    rA1;
      L     #Set001.OutAlarmNumberMOZF;
      T     #OutAlarmNrMOZF;
//--- keep old alarm number  MYFC ------------
rA1:  L     0;
      L     #Set001.OutAlarmNumberMYFC;
      ==I;
      =     #Par.OutFlags.OutNoAlarmMYFC;
//      U     #OutFlags.OutNoAlarmMYFC
      A     #Par.OutFlags.OutRelevantFaultMYFC;
      AN    #Par.OutFlags.OutTestNewAlarm;
      AN    #tmpLocal;
      AN    #InManual;
      JC    r000;
      L     #Set001.OutAlarmNumberMYFC;
      T     #OutAlarmNrMYFC;
//================================================
r000: A     #tmpCallBackFuction;
      BEC;
rEnd: NOP   0;
NETWORK
TITLE =  Read from Queue (****Opto22 ****)
////*************************************************
////***             O P T O 22                    ***
////*************************************************
//
      A     #Par.ParDP;
      JC    Ct00;
      OPN   DB [#tmpComDB];
      L     #Par.ParLCIdx;
      T     DBW 34;	//COM.Element.Index;
      L     1;	//Read LC data
      T     DBW 0;	//COM.CODE;
      CDB;
      UC    "GCS7_RS485Ctrl";
      CDB;
      L     #tmpFBNO;
      T     DBW 52;	//COM.LC0.FBNO;   
      L     DINO;
      T     DBW 54;	//COM.LC0.DINO;
      TAR2  DBD 56;	//COM.LC0.AddrDyn;        
      L     #Par.ParObjectNo;
      T     DBD 60;	//COM.LC0.AddrPara;       
      L     #Par.ParLCAddr;
      T     DBD 64;	//COM.Telegram.LCAddr;
Ct00: NOP   0;
NETWORK
TITLE =  All State Init
//===Clear tmp Variable
      NOP   0;
//===Global Group Orders===
// -->[2.2]
      A     "GCS7_Gr_OutManualOn";	//Global.OutManualOn
      S     #InManual;
      A     "GCS7_Gr_OutManualOff";	//Global.OutManualOff
      R     #InManual;
      A     #InManual;
      S     "GCS7_Gr_InManual";	//Global.InManualMode
// <--[2.2]
//--tmpEnable
      A(;
      AN    #InManual;
      ON    #Par.ParManual;
      A     #InEnable;
      AN    #tmpLocal;
      O;
      A     #InManual;
      A     #Par.ParManual;
      );
      AN    #InHWStop;
      AN    #InDPFault;
      AN    #CmdOff;
      =     #tmpEnable;
//---Report is on---
      O     "GCS7_Gr_OutReportAll";	//---Global OutReportAll
      O     #InReport;
      =     #tmpReport;
//---FaultReset is on---
      A     "GCS7_Gr_OutFaultReset";	//Gr.OutFaultReset
      S     #CmdFaultReset;
//---Check mode
      AN    #InManualWaterControl;
      A     #Par.Status.Manual;
      O;
      AN    #InManualWaterControl;
      AN    #InLocalWaterControl;
      AN    #Par.Status.Remote;
      =     #OutFaultMode;
//---ComFault
      A     #Par.OutFlags.OutComFaultRead;
      O     #Par.OutFlags.OutComFaultSend;
      A     #Par.ParDP;
      O;
      AN    #Par.ParDP;
      A     #OutFaultCom;
      =     #OutFaultCom;
//===Prepare Alarm Flags=========================== 
      LAR1  P##tmpFilter;
      L     #OutAlarmNrMYFC;
      +AR1;
      L     #OutAlarmNrMYFC;
      L     0;
      <>I;
      AN    L [AR1,P#0.0];	//#tmpFilter[OutAlarmNumberMYFC]
      =     #Par.OutFlags.OutRelevantFaultMYFC;
      LAR1  P##tmpFilter;
      L     #OutAlarmNrMOZF;
      +AR1;
      L     #OutAlarmNrMOZF;
      L     0;
      <>I;
      AN    L [AR1,P#0.0];	//#tmpFilter[OutAlarmNumberMOZF]
      =     #Par.OutFlags.OutRelevantFaultMOZF;
      A     #Par.OutFlags.OutRelevantFaultMYFC;
      O     #Par.OutFlags.OutRelevantFaultMOZF;
      =     #OutFaultRelevant;
      L     #OutAlarmNrMYFC;
      L     0;
      <>I;
      AN    #Par.ParMOZF;
      O(;
      L     #OutAlarmNrMOZF;
      L     0;
      <>I;
      );
      AN    #OutFaultRelevant;
      =     #OutWarning;
      A     #OutFaultRelevant;
      O     #OutFaultCom;
      O     #OutWrongValue;
      AN    #InManualWaterControl;
      O     #OutFaultMode;
      O(;	//[1.1]
      AN    #Par.Status.RemoteControlDP;	//[1.1]
      AN    #InLocalWaterControl;	//[1.1]
      AN    #InManualWaterControl;	//[1.1]
      A     #Par.ParDP;	//[1.1]
      );	//[1.1]
      AN    #InHWStop;
      AN    #InDPFault;
      AN    #tmpLocal;
      =     #tmpFault;
//---CmdNewJob
      AN    #CmdNewJob;
      JC    in2;
      R     #CmdNewJob;
      L     0;
      T     #OutTotalProduct;
      T     #OutTotalWater;
in2:  NOP   0;
NETWORK
TITLE = States
//===State machine===
      A     #StStopped;
      JC    S0;
      A     #StDosing;
      JC    S2;
      A     #StWaiting;
      JC    S5;
      A     #StStarting;
      JC    S1;
      A     #StStopping;
      JC    S3;
      A     #StFault;
      JC    S4;
      JU    xxS0;	//Init
NETWORK
TITLE =  StStopped
//Automatic fault reset
xxS0: S     #StStopped;	//Init
      L     B#(4, 91);	// MessageClass Info stopped
      A     #tmpReport;
      JC    LOG;
//---Condition for StFault
S0:   A     #tmpFault;
      R     #StStopped;
      JC    xxS4;	//-->StFault
//---Condition for StStarting
      A     #CmdNext;
      AN    #InManual;
      O     #CmdOn;
      A     #tmpEnable;
      R     #StStopped;
      JC    xxS1;
      JU    OUT;
NETWORK
TITLE =  StStarting
//Automatic fault reset
xxS1: S     #StStarting;
      L     #Par.ParMonTime;
      T     #Par.OutMonTime;
//---Condition for StFault
S1:   A     #tmpFault;
      R     #StStarting;
      JC    xxS4;	//-->StFault
//---Monitoring Starting
      AN    "GCS7_Gr_OutTick200ms";
      L     #Par.OutMonTime;
      JC    S1J1;
      +     -2;
      T     #Par.OutMonTime;
S1J1: L     0;
      <=I;	//---Condition for StStarted
      R     #StStarting;
      S     #tmpFaultMonitoringStart;
      JC    xxS4;	//---Transition -> StFault
//---Condition for StStopping
      AN    #tmpEnable;
      R     #StStarting;
      JC    xxS3;	//-->StStopping
//---Condition for StEnabled
      A     #Par.Status.Enable24V;
      A     #Par.Status.Active;
      AN    #InManualWaterControl;
      O;
      A     #OutpEnable;
      A     #InManualWaterControl;
      R     #StStarting;
      JC    xxS5;	//-->StWaiting
      JU    OUT;
NETWORK
TITLE =  StDosing
xxS2: S     #StDosing;
      L     B#(4, 92);	// MessageClass Info stopped
      A     #tmpReport;
      JC    LOG;
      JU    OUT;
//Condition for StFault
S2:   A     #tmpFault;
      R     #StDosing;
      JC    xxS4;	//--> StFault
//---Condition for StStopping
      AN    #Par.Status.Dosing;
      AN    #InManualWaterControl;
      ON    #tmpEnable;
      R     #StDosing;
      JC    xxS5;	//-->StWaiting
      JU    OUT;
NETWORK
TITLE =  StStopping
//Automatic fault reset
xxS3: S     #StStopping;
      L     #Par.ParMonTime;
      T     #Par.OutMonTime;
//---Condition for StFault
S3:   A     #tmpFault;
      R     #StStopping;
      JC    xxS4;	//-->StFault
//---Condition for StStopping
      AN    #Par.Status.Enable24V;
      AN    #InManualWaterControl;
      O;
      AN    #OutpEnable;
      A     #InManualWaterControl;
      O     #InHWStop;
      O     #InDPFault;
      O     #InLocal;	// [2.3]
      R     #StStopping;
      JC    xxS0;	//-->StStopped
//---Monitoring Stoopin
      AN    "GCS7_Gr_OutTick200ms";
      L     #Par.OutMonTime;
      JC    S3J1;
      +     -2;
      T     #Par.OutMonTime;
S3J1: L     0;
      <=I;
      R     #StStopping;
      S     #tmpFaultMonitoringStop;
      JC    xxS4;	//---Transition -> StFault
      JU    OUT;
NETWORK
TITLE =  StWaiting
xxS5: S     #StWaiting;
      L     B#(4, 93);	// MessageClass Info stopped
      A     #tmpReport;
      JC    LOG;
//---Condition for StFault
S5:   A     #tmpFault;
      R     #StWaiting;
      JC    xxS4;	//--> StFault
//---Condition for StDosing
      A     #OutpEnable;
      A     #InManualWaterControl;
      A     #tmpEnable;
      O;
      A     #Par.Status.Dosing;
      AN    #InManualWaterControl;
      A     #tmpEnable;
      R     #StWaiting;
      JC    xxS2;	//-->StDosing
//---Condition for StStopping
      AN    #tmpEnable;
      ON    #Par.Status.Enable24V;
      ON    #Par.Status.Active;
      R     #StWaiting;
      JC    xxS3;	//-->StStopping
      JU    OUT;
NETWORK
TITLE =  StFault
S4:   A     #Par.OutFlags.OutTestNewAlarm;
      O     #InManualWaterControl;
      AN    #tmpFault;
      O     #tmpLocal;
      JC    S4S5;
//---Monitoring Alarm reset
      AN    "GCS7_Gr_OutTick200ms";
      ON    #Par.OutFlags.OutTestNewAlarm;	// Relog fault
      L     #Par.OutMonTime;
      JC    S4J1;
      +     -2;
      T     #Par.OutMonTime;
S4J1: L     0;
      <=I;	//---Condition for  Relog fault
      A     #Par.OutFlags.OutTestNewAlarm;	// Relog fault
      A     #tmpFault;
      JC    xxS4;
      JU    OUT;
//Transition to StStopped 
S4S5: S     #StStopping;
      R     #StFault;
      L     B#(3, 0);	//Message ('fault cancelled')
      JU    LOG;
NETWORK
TITLE = LOG
//91   = StStopped
//92   = StDosing
//93   = StWaiting
//94   = Timeout starting
//95   = Timeout stopping
//96   = Communication fault
//97   = FaultManualMode
//98   = FaultLocalMode
//99   = FaultWrongValue
//
xxS4: A     #StFault;	// 2.1: Fault flag only when transition -> StFault
      JC    S4J2;
      S     "GCS7_Gr_InFaultFlag";	// 2.1: Gr.InFaultFlag
      CALL  "SYS_Horn_Code" (
           FcCode                   := 1,
           ParObjectType            := 1034,
           ParObjectNo              := #Par.ParObjectNo,
           ParHornCode              := #Par.ParHornCode);
S4J2: SET;	// 2.1:
      S     #StFault;
      R     #Par.OutFlags.OutTestNewAlarm;
      L     50;	// [1.2] 5s for retry fault
      T     #Par.OutMonTime;	// [1.2]
//Alarm Moonitoring
      A     #tmpFaultMonitoringStart;
      L     B#(1, 94);	// MessageClass Error fault starting
      JC    LOG;
      A     #tmpFaultMonitoringStop;
      L     B#(1, 95);	// MessageClass Error fault starting
      JC    LOG;
//Alarm Communication
      L     B#(1, 96);
      A     #OutFaultCom;
      JC    LOG;
//Alarm Message MYFC
      AN    #Par.OutFlags.OutRelevantFaultMYFC;
      JC    LoF;
      L     #OutAlarmNrMYFC;
      L     B#(1, 0);
      OW;
      JU    LOG;	//Alarms 11..80
//Alarm Message MOZF
LoF:  AN    #Par.OutFlags.OutRelevantFaultMOZF;
      JC    LoM;
      L     #OutAlarmNrMOZF;
      L     B#(1, 0);
      OW;
      JU    LOG;	//Alarms 11..80
// Alarm Mode
LoM:  L     B#(1, 97);
      A     #OutFaultMode;
      A     #Par.Status.Manual;
      JC    LOG;
      L     B#(1, 98);
      A     #OutFaultMode;
      AN    #Par.Status.Remote;
      JC    LOG;
//Alarm 'fault DP Mode                                                       
      L     B#(1, 90);	// Message ('fault DP Mode')   //[1.1]
      AN    #Par.Status.RemoteControlDP;	//[1.1]
      AN    #InLocalWaterControl;	//[1.1]
      AN    #InManualWaterControl;	//[1.1]
      A     #Par.ParDP;	//[1.1]
      JC    LOG;	//[1.1]
//Wrong Value
      A     #OutWrongValue;
      L     B#(1, 99);	// Message ('fault wrong value')  //[1.4]
      JC    LOG;
//Alarm Communication
      L     B#(1, 96);	//COM communication
      JU    LOG;
LOG:  A     #Par.ParLogOff;	//---Set LOG Message
      JC    OUT;
      T     #tmpLOGvalue;
      L     B#(0, 255);	//COM communication
      AW;
      T     #OutAlarmNrLog;
      CALL  "GCS7_LogConvert" (
           ObjectNo                 := #Par.ParObjectNo,
           MsgType                  := #Par.ParMsgType,
           ClassMsgTxt              := #tmpLOGvalue,
           OType                    := 1034);	//LOG Message Converter / Entry / Contains Class and TextNo
NETWORK
TITLE = Global End
OUT:  SET;	//---Clear all commands
      R     #CmdNext;
      R     #CmdOn;
      R     #CmdOff;
      AN    #StFault;
      R     #Par.OutFlags.OutTestNewAlarm;
      A     #StStarting;
      O     #StWaiting;
      O     #StDosing;
      =     #OutpEnable;
//--Output for group 
      AN    #InLocal;
      O     #InManual;
      A     #InDPFault;
      S     "GCS7_Gr_InDPFault";
      AN    #InLocal;
      O     #InManual;
      A     #InHWStop;
      S     "GCS7_Gr_InHWStop";
NETWORK
TITLE = State Code
      AN    #StStopped;
      JC    sc3;
      L     41;	//Code: StStopped HWStop
      A     #InHWStop;
      JC    STC;
      L     51;	//Code: StStopped DPStop
      A     #InDPFault;
      JC    STC;
      L     1;	//Code: StStopped
      JU    STC1;
sc3:  L     6;	//Code: StEmptying  [2.0]
      A     #StDosing;	//                  [2.0]
      O     #StWaiting;	//                  [2.1]
      A     #InRestdischarge;	//                  [2.0]
      AN    #InManualWaterControl;	//                  [2.0]
      JC    STC1;
      L     3;	//Code: StDosingAuto
      A     #StDosing;
      AN    #InManualWaterControl;
      JC    STC1;
      L     4;	//Code: StDosingManual
      A     #StDosing;
      JC    STC1;
      L     5;	//Code: StWaiting
      A     #StWaiting;
      JC    STC1;
      L     2;	//Code: StStarting
      A     #StStarting;
      JC    STC1;
      L     7;	//Code: StStopping
      A     #StStopping;
      JC    STC1;
      L     32;	//Code: fault
      JU    STC;
//Test Warning : StCode = StCode+10
STC1: AN    #OutWarning;
      JC    STC;
      +     10;	// StCode = StCode+10
STC:  L     #StCode;	//Old state code
      TAK;
      T     #StCode;	//Save state code
      <>I;
      L     3;	//Load code for CBit methode
      CC    "SYS_CBitCtrl";
NETWORK
TITLE = Prepare Command for LC (** DP **)
////*************************************************
////***            DP Communication              ***
////*************************************************
//
      AN    #Par.ParDP;
      JC    sEnd;
//==============================
      A     #InRestdischarge;	// [2.0]
      =     #Par.Command.InRestdischarge;	//[2.0]
      A     #Par.Status.AcceptNewSendData;
      A     #Par.Command.ResetAlarm;
      R     #Par.Command.ResetAlarm;
      S     #Par.OutFlags.OutFaultResetDone;
      A     #CmdFaultReset;
      AN    #Par.Status.AcceptNewSendData;
      R     #CmdFaultReset;
      S     #Par.Command.ResetAlarm;
//==============================
      A     #Par.Status.NewDataReady;
      =     #Par.Command.AcceptNewDataReady;
//==============================
      SET;
      =     #Par.Command.CommandReady;
//==============================
      A     #Par.Status.NewRcvData;
      =     #Par.Command.AcceptNewRcvData;
//==============================
      AN    #Par.Status.AcceptNewSendData;
      =     #Par.Command.NewSendData;
NETWORK
TITLE = Send Data (**DP**)
////*************************************************
////***            DP Communication              ***
////*************************************************
//
//======================================================
//Test Send Dataset 000 done
      L     #DPData.NrSndDataSet;
      L     0;
      <>I;
      JC    s128;
      JU    S128;	//-->send 128
//------------------------------------------------
//Test Send Dataset 128 done
s128: L     #DPData.NrSndDataSet;
      L     128;
      <>I;
      JC    s136;
      A     #Par.Status.WrongValue;
      =     #OutWrongValue;
      JU    S136;	//-->Send 136
//------------------------------------------------
//Test Send 136 done
s136: L     #DPData.NrSndDataSet;
      L     136;
      <>I;
      JC    S000;
      A     #Par.Status.WrongValue;
      =     #OutWrongValue;
      JU    S128;	//-->Send 128
//==================================================
//Send Dataset 128
S128: AN    #Par.ParMOZF;
      JC    S136;	//-->Send 136
      L     128;
      T     #DPData.NrSndDataSet;
      L     0;
      T     #DPData.IdxSndDataSet;
      L     #InMoisture;
      SLD   16;
      T     #DPData.Data[1];
      L     0;
      T     #DPData.Data[2];
      T     #DPData.Data[3];
      T     #DPData.Data[4];
      JU    sndD;
//======================================================
//Send Dataset 136
S136: A     #Par.ParMOZF;
      JC    S000;
      L     136;
      T     #DPData.NrSndDataSet;
      L     0;
      T     #DPData.IdxSndDataSet;
      L     #InMoisture;
      T     #Set136.InMoistureNom;
      L     #InOffsetMoisture;
      T     #Set136.InMoistureOffset;
      L     #InDosingMax;
      T     #Set136.InDosingMax;
      L     #InProductGroup;
      T     #Set136.InProductGroup;
      L     0;
      T     #Set136.Spare17;
      L     0;
      T     #Set136.Spare18;
      L     0;
      T     #Set136.Spare22;
      CALL  "SIEMENS_BLKMOV" (
           SRCBLK                   := #Set136,
           RET_VAL                  := #tmpReturn,
           DSTBLK                   := #DPData.Data);
      JU    sndD;
//======================================================
//Send Dataset 0
S000: L     0;
      T     #DPData.NrSndDataSet;
      L     0;
      T     #DPData.IdxSndDataSet;
//======================================================
//Send to DP
sndD: CALL  "SIEMENS_BLKMOV" (
           SRCBLK                   := #Par.Command,
           RET_VAL                  := #tmpReturn,
           DSTBLK                   := #DPData.StatusCommand);
      A     #InSimulation;
      JC    sSim;
      CALL  "SIEMENS_DPWR_DAT" (
           LADDR                    := #tmpAddr,
           RECORD                   := #DPData,
           RET_VAL                  := #tmpReturn);
      L     #tmpReturn;
      L     0;
      <>I;
      =     #Par.OutFlags.OutComFaultSend;
      JU    sEnd;
//write to Simulation
sSim: R     #Par.OutFlags.OutComFaultSend;
      A     "GCS7_Gr_SimDPtoImage";
      L     P#Q 0.0;
      JC    rDB2;
      OPN   "TEST_IOSimuliOutput";
      L     P#DBX 0.0;
rDB2: L     #Par.ParIOByteNr;
      SLD   3;
      +D;
      LAR1;
      L     #DPData.StatusCommand;
      T     D [AR1,P#0.0];
      L     #DPData.NrSndDataSet;
      T     B [AR1,P#4.0];
      L     #DPData.IdxSndDataSet;
      T     B [AR1,P#5.0];
      L     #DPData.NrRcvDataSet;
      T     B [AR1,P#6.0];
      L     #DPData.IdxRcvDataSet;
      T     B [AR1,P#7.0];
      L     #DPData.Data[1];
      T     D [AR1,P#8.0];
      L     #DPData.Data[2];
      T     D [AR1,P#12.0];
      L     #DPData.Data[3];
      T     D [AR1,P#16.0];
      L     #DPData.Data[4];
      T     D [AR1,P#20.0];
sEnd: NOP   0;
NETWORK
TITLE = Communication
////*************************************************
////***             O P T O 22                    ***
////*************************************************
//
      A     #Par.ParDP;
      JC    com0;
      L     'C';
      AN    #Par.ParMOZF;
      JC    com2;
      L     'F';
com2: S     DBX 50.0;	//COM.LC0.CmdPut ;
      T     DBB 51;	//COM.LC0.Command;
com0: NOP   0;
NETWORK
TITLE =  Store LC data (***OPTO22 **)
////*************************************************
////***             O P T O 22                    ***
////*************************************************
//
      A     #Par.ParDP;
      BEC;
      L     #Par.ParLCIdx;
      T     DBW 34;	//COM.Element.Index; 
      L     2;	//Store LC data
      T     DBW 0;	//COM.CODE;
      CDB;
      UC    "GCS7_RS485Ctrl";
      CDB;
      BEU;
NETWORK
TITLE = Calculate Total Weight
END_FUNCTION_BLOCK

FUNCTION_BLOCK "GCS7_E_MDDx"	// FB 35
TITLE = MDDx Serial Communication
//  
//COPYRIGHT:    (C) 1998  BUHLER AG, CH-9240 UZWIL, SWITZERLAND
//
//PRODUCT:      GCS7
//
//TITLE:        Element Control MDDx Serial Communication
//              GCPROVB Revision 11   
//
//-------------------------------------------------------------------------
//
//IDENT:        AUTHOR:             DEPT:                      DATE:
//
//FB35.4.0      A. Egli             CT3                        18-Mai-2004
//              MDDO/M
//FB35.3.1      A. Egli             CT3                        02-Sep-2003
//              Fault at calculation of address of parameter 
//FB35.3.0      A. Egli             CT3                        17-Jun-2002
//              New Release with one block 
//FB35.2.2      A. Egli             CT3                        17-Mar-2000
//              Length for answer telegram
//FB35.2.1      S. Kalberer         CT3                        19-Jan-2000
//              LOG and fault reset by warning but not local mode
//FB35.2.0      S. Kalberer         CT3                        06-Dec-1999
//              New alarms 7,8,12,28-31 adapted to LOG
//              Set Horn on transition to fault or warning and not InLocal
//              No cyclic command "S" sending (UDT20351 has changed!)
//FB35.1A       S. Kalberer         CT3                        24-Sep-1999
//              Release in S7
//
//-------------------------------------------------------------------------
//
//PURPOSE:      MANUAL : see [MDDENMAN]
//
//RESTRICTIONS: S7
//              ACCU2: Pointer to dynamic datas of the element
//              ACCU1: Pointer to parameter datas of the element
//              tmpFault and tmpWarning may be set together!
//
//-------------------------------------------------------------------------
//=======================================================
//Log Message: 
//------------------------------------------------------
//  1  EPROM wrong checksum         = #Par.Par.OutLCAlarm.CheckSumFault
//  2  RAM test fault               = #Par.Par.OutLCAlarm.RAMTestFault
//  3  Operation fault              = #Par.Par.OutLCAlarm.OperationFault
//  4  Watchdog                     = #Par.Par.OutLCAlarm.WatchDog
//  5  Memory lost                  = #Par.Par.OutLCAlarm.MemoryLost
//  6  No communication with grinding gap print
//                                  = #Par.Par.OutLCAlarm.GrindGapPrint
//  7  ERR 7                        = #Par.Par.OutLCAlarm.ERR0007
//  8  ERR 8                        = #Par.Par.OutLCAlarm.ERR0008
//  9  Fault cancelled
// 10  MDDx communication fault
// 11  Dry running of grinding rolls= #Par.Par.OutLCAlarm.GrindRollsDryRun
// 12  ERR 12                       = #Par.Par.OutLCAlarm.ERR0012
// 13  Standstill of feed rolls     = #Par.Par.OutLCAlarm.FeedRollsStandstill
// 14  Standstill of grinding rolls = #Par.Par.OutLCAlarm.GrindRollsStandstill
// 15  Standstill of lower grinding rolls
//                                 = #Par.Par.OutLCAlarm.GrindRollsLowStandstill
// 16 Overload of main motor       = #Par.Par.OutLCAlarm.MotorOverload;
// 17 Overload of lower motor      = #Par.Par.OutLCAlarm.MotorLowOverload;
// 18 Grinding gap fault           = #Par.Par.OutLCAlarm.GrindGapFault;
// 19 Lower grinding gap fault     = #Par.Par.OutLCAlarm.GrindGapLowFault;
// 20 Product registration fault   = #Par.Par.OutLCAlarm.ProdRegistrationFault;
// 21 Grinding gap no increment    = #Par.Par.OutLCAlarm.GrindGapNoIncr;
// 22 Lower grinding gap no increment
//                                 = #Par.Par.OutLCAlarm.GrindGapLowNoIncr;
// 23 HL inlet                     = #Par.Par.OutLCAlarm.HLInlet;
// 24 HL outlet                    = #Par.Par.OutLCAlarm.HLOutlet;
// 25 HL backup left               = #Par.Par.OutLCAlarm.HLBackUpLeft;
// 26 HL backup right              = #Par.Par.OutLCAlarm.HLBackUpRight;
// 27 Emergency stop was pressed   = #Par.Par.OutLCAlarm.EmergencyStop;
// 28 Product is full or the feed roll maximum speed
//                                 = #Par.Par.OutLCAlarm.InletProductFullRpnmax
// 29 Not enough product in the inlet
//                                 = #Par.Par.OutLCAlarm.InletNotEnoughProduct
// 30 ERR 30                       = #Par.Par.OutLCAlarm.ERR0030
// 31 ERR 31                       = #Par.Par.OutLCAlarm.ERR0031
//
//=======================================================
//StCode:  State               
//------------------------------------------------------
//
//32  StFault                 
// 3  StOk                    
// 5  StWarning               
//45  StWarning.HWStop               StStopped + InHWStop 
//55  StWarning.DPFault              StStopped + DPFault
//
AUTHOR : EA
FAMILY : GCS7LL
NAME : MDDxSer
VERSION : 4.0
VAR
  StCode : INT ;	//Element state code
  InEnableEngage : BOOL ;	//Signal to engage the rolls
  InRestdischarge : BOOL ;	//Signal to activate restdischarge mode
  spare0202 : BOOL ;
  spare0203 : BOOL ;
  CmdNewValue : BOOL ;
  spare0205 : BOOL ;
  spare0206 : BOOL ;
  spare0207 : BOOL ;
  spare0300 : BOOL ;
  spare0301 : BOOL ;
  spare0302 : BOOL ;
  CmdFaultReset : BOOL ;	//Command to reset fault
  InLocal : BOOL ;	//1= Local mode (no fault by start with service switch)
  spare0305 : BOOL ;
  spare0306 : BOOL ;
  spare0307 : BOOL ;
  InHWStop : BOOL ;	//HW stop is detected, no fault
  InDPFault : BOOL ;	//DP-Fault is detected, no fault
  OutComFault : BOOL ;	//Communication fault
  OutFaultResetDone : BOOL ;	//Aux. signal fault reset done
  spare0404 : BOOL ;
  spare0405 : BOOL ;
  spare0406 : BOOL ;
  spare0407 : BOOL ;
  spare0500 : BOOL ;
  spare0501 : BOOL ;
  StOk : BOOL ;	//Element is ok
  spare0503 : BOOL ;
  StFault : BOOL ;	//Element has a communication or device fault
  StWarning : BOOL ;	//Element is in local mode or has a warning fault
  OutFeedRollSpeed : INT ;	//Is read from LC [0..0500 RPM]
  OutFeedRollStatus : INT ;	//Is read from LC [0..9999]
  OutRollsUpCurrent : INT ;	//Is read from LC [0.1 A]
  OutRollsLowCurrent : INT ;	//Is read from LC [0.1 A]
  OutRollsUpLoad : INT ;	//Is read from LC [%]
  OutRollsLowLoad : INT ;	//Is read from LC [%]
  OutGrindGapStatus : INT ;	//Is read from LC [0..9999]
  OutAlarmNr : INT ;	//Is read from LC [0..9999]
  spare2200 : INT ;	//Is read from LC [0..9999]
  OutLCState : STRUCT 	//Is read from LC [Bit]
   spare00 : BYTE ;
   RollStandMDDM : BOOL ;	//Roll stand type: 0=MDDO / 1=MDDM
   HLInlet : BOOL ;	//HL inlet: 1=Covered
   HLOutlet : BOOL ;	//HL outlet: 1=Covered
   HLBackUp : BOOL ;	//HL backup: 1=Covered
   RestDischarge : BOOL ;	//Restdischarge: 1=Active
   Disengaged : BOOL ;	//Rolls: 1=Disengaged
   ManDisengaged : BOOL ;	//Rolls manually disengaged: 1=Manually disengaged
   spare17 : BOOL ;
  END_STRUCT ;
  spare2600 : INT ;
  spare2800 : INT ;
  OutAlarmNrLog : INT ;	//Last textnumber send to log
  InGapData : STRUCT 	//Only without MDEF
   Spare0 : INT ;
   GapTopLeft : INT ;	//de:  Sollwert Mahlspalt oben links
   GapTopRight : INT ;	//de:  Sollwert Mahlspalt oben rechts
   GapBottomLeft : INT ;	//de:  Sollwert Mahlspalt unten links
   GapBottomRight : INT ;	//de:  Sollwert Mahlspalt unten rechts
   GapAdjustment : INT ;
  END_STRUCT ;
  OutGapData : STRUCT 	//Only without MDEF
   Spare0 : INT ;
   GapTopLeftNom : INT ;	//de:  Sollwert Mahlspalt oben links
   GapTopRightNom : INT ;	//de:  Sollwert Mahlspalt oben rechts
   GapBottomLeftNom : INT ;	//de:  Sollwert Mahlspalt unten links
   GapBottomRightNom : INT ;	//de:  Sollwert Mahlspalt unten rechts
   GapTopLeftAc : INT ;	//de:  Istwert Mahlspalt oben links
   GapTopRightAc : INT ;	//de:  Istwert Mahlspalt oben rechts
   GapBottomLeftAc : INT ;	//de:  Istwert Mahlspalt unten links
   GapBottomRightAc : INT ;	//de:  Istwert Mahlspalt unten rechts
   GapAdjustment : INT ;	//0=Off;1=Manual;2=Automatic;3=Referencing;4=Aligment;5=Save
  END_STRUCT ;
  Par : STRUCT
   ParObjectNo : INT ;	//Is used for communication with PC, e.g. for message
   ParMsgType : INT ;	//Is used for message (translation of state)
   ParHornCode : INT ;	//Is used by horn module
   ParLogOff : BOOL ;	//Report is off
   spare0401 : BOOL ;
   ParWarning : BOOL ;	//Warning mode for communication fault (see OutComFault)
   ParNoMDEF : BOOL ;	//1=No MDEF : read and write of grinding gap data
   spare04041 : BOOL ;
   ParFilter : STRUCT 	//Filter to alarm 1=Ignore alarm
    spare00 : BOOL ;
    CheckSumFault : BOOL ;	//ERR  1 - EPROM wrong checksum
    RAMTestFault : BOOL ;	//ERR  2 - RAM test fault
    OperationFault : BOOL ;	//ERR  3 - Operation fault
    WatchDog : BOOL ;	//ERR  4 - Watchdog
    MemoryLost : BOOL ;	//ERR  5 - Memory lost
    GrindGapPrint : BOOL ;	//ERR  6 - No communication with grinding gap print
    ERR0007 : BOOL ;	//ERR  7 - not defined
    ERR0008 : BOOL ;	//ERR  8 - not defined
    ERR0009 : BOOL ;	//ERR  9 - not defined (reserved PLC message)
    ERR0010 : BOOL ;	//ERR 10 - not defined (reserved PLC message)
    GrindRollsDryRun : BOOL ;	//ERR 11 - Dry running of grinding rolls
    ERR0012 : BOOL ;	//ERR 12 - not defined
    FeedRollsStandstill : BOOL ;	//ERR 13 - Standstill of feed rolls
    GrindRollsStandstill : BOOL ;	//ERR 14 - Standstill of grinding rolls
    GrindRollsLowStandstill : BOOL ;	//ERR 15 - Standstill of lower grinding rolls
    MotorOverload : BOOL ;	//ERR 16 - Overload of main motor
    MotorLowOverload : BOOL ;	//ERR 17 - Overload of lower motor
    GrindGapFault : BOOL ;	//ERR 18 - Grinding gap fault
    GrindGapLowFault : BOOL ;	//ERR 19 - Lower grinding gap fault
    ProdRegistrationFault : BOOL ;	//ERR 20 - Product registration fault
    GrindGapNoIncr : BOOL ;	//ERR 21 - Grinding gap no increment
    GrindGapLowNoIncr : BOOL ;	//ERR 22 - Lower grinding gap no increment
    HLInlet : BOOL ;	//ERR 23 - HL inlet
    HLOutlet : BOOL ;	//ERR 24 - HL outlet
    HLBackUpLeft : BOOL ;	//ERR 25 - HL backup left
    HLBackUpRight : BOOL ;	//ERR 26 - HL backup right
    EmergencyStop : BOOL ;	//ERR 27 - Emergency stop was pressed
    InletProductFullRpnmax : BOOL ;	//ERR 28 - Product is full or the feed roll is rotating at maximum speed
    InletNotEnoughProduct : BOOL ;	//ERR 29 - Not enough product in the inlet
    ERR0030 : BOOL ;	//ERR 30 - not defined
    ERR0031 : BOOL ;	//ERR 31 - not defined
   END_STRUCT ;
   ParFilterWarning : STRUCT 	//Filter to set alarm type (0=Fault;Suspend/1=Warning)
    spare00 : BOOL ;
    CheckSumFault : BOOL ;	//ERR  1 - EPROM wrong checksum
    RAMTestFault : BOOL ;	//ERR  2 - RAM test fault
    OperationFault : BOOL ;	//ERR  3 - Operation fault
    WatchDog : BOOL ;	//ERR  4 - Watchdog
    MemoryLost : BOOL ;	//ERR  5 - Memory lost
    GrindGapPrint : BOOL ;	//ERR  6 - No communication with grinding gap print
    ERR0007 : BOOL ;	//ERR  7 - not defined
    ERR0008 : BOOL ;	//ERR  8 - not defined
    ERR0009 : BOOL ;	//ERR  9 - not defined (reserved PLC message)
    ERR0010 : BOOL ;	//ERR 10 - not defined (reserved PLC message)
    GrindRollsDryRun : BOOL ;	//ERR 11 - Dry running of grinding rolls
    ERR0012 : BOOL ;	//ERR 12 - not defined
    FeedRollsStandstill : BOOL ;	//ERR 13 - Standstill of feed rolls
    GrindRollsStandstill : BOOL ;	//ERR 14 - Standstill of grinding rolls
    GrindRollsLowStandstill : BOOL ;	//ERR 15 - Standstill of lower grinding rolls
    MotorOverload : BOOL ;	//ERR 16 - Overload of main motor
    MotorLowOverload : BOOL ;	//ERR 17 - Overload of lower motor
    GrindGapFault : BOOL ;	//ERR 18 - Grinding gap fault
    GrindGapLowFault : BOOL ;	//ERR 19 - Lower grinding gap fault
    ProdRegistrationFault : BOOL ;	//ERR 20 - Product registration fault
    GrindGapNoIncr : BOOL ;	//ERR 21 - Grinding gap no increment
    GrindGapLowNoIncr : BOOL ;	//ERR 22 - Lower grinding gap no increment
    HLInlet : BOOL ;	//ERR 23 - HL inlet
    HLOutlet : BOOL ;	//ERR 24 - HL outlet
    HLBackUpLeft : BOOL ;	//ERR 25 - HL backup left
    HLBackUpRight : BOOL ;	//ERR 26 - HL backup right
    EmergencyStop : BOOL ;	//ERR 27 - Emergency stop was pressed
    InletProductFullRpnmax : BOOL ;	//ERR 28 - Product is full or the feed roll is rotating at maximum speed
    InletNotEnoughProduct : BOOL ;	//ERR 29 - Not enough product in the inlet
    ERR0030 : BOOL ;	//ERR 30 - not defined
    ERR0031 : BOOL ;	//ERR 31 - not defined
   END_STRUCT ;
   ParComDB : INT ;	//Communication DB
   ParLCIdx : INT ;	//Index of data record
   ParLCAddr : INT ;	//Address of LC
   OutLCAlarm : STRUCT 	//Alarm bit mask of OutAlarmNumber
    spare00 : BOOL ;
    CheckSumFault : BOOL ;	//ERR  1 - EPROM wrong checksum
    RAMTestFault : BOOL ;	//ERR  2 - RAM test fault
    OperationFault : BOOL ;	//ERR  3 - Operation fault
    WatchDog : BOOL ;	//ERR  4 - Watchdog
    MemoryLost : BOOL ;	//ERR  5 - Memory lost
    GrindGapPrint : BOOL ;	//ERR  6 - No communication with grinding gap print
    ERR0007 : BOOL ;	//ERR  7 - not defined
    ERR0008 : BOOL ;	//ERR  8 - not defined
    ERR0009 : BOOL ;	//ERR  9 - not defined (reserved PLC message)
    ERR0010 : BOOL ;	//ERR 10 - not defined (reserved PLC message)
    GrindRollsDryRun : BOOL ;	//ERR 11 - Dry running of grinding rolls
    ERR0012 : BOOL ;	//ERR 12 - not defined
    FeedRollsStandstill : BOOL ;	//ERR 13 - Standstill of feed rolls
    GrindRollsStandstill : BOOL ;	//ERR 14 - Standstill of grinding rolls
    GrindRollsLowStandstill : BOOL ;	//ERR 15 - Standstill of lower grinding rolls
    MotorOverload : BOOL ;	//ERR 16 - Overload of main motor
    MotorLowOverload : BOOL ;	//ERR 17 - Overload of lower motor
    GrindGapFault : BOOL ;	//ERR 18 - Grinding gap fault
    GrindGapLowFault : BOOL ;	//ERR 19 - Lower grinding gap fault
    ProdRegistrationFault : BOOL ;	//ERR 20 - Product registration fault
    GrindGapNoIncr : BOOL ;	//ERR 21 - Grinding gap no increment
    GrindGapLowNoIncr : BOOL ;	//ERR 22 - Lower grinding gap no increment
    HLInlet : BOOL ;	//ERR 23 - HL inlet
    HLOutlet : BOOL ;	//ERR 24 - HL outlet
    HLBackUpLeft : BOOL ;	//ERR 25 - HL backup left
    HLBackUpRight : BOOL ;	//ERR 26 - HL backup right
    EmergencyStop : BOOL ;	//ERR 27 - Emergency stop was pressed
    InletProductFullRpnmax : BOOL ;	//ERR 28 - Product is full or the feed roll is rotating at maximum speed
    InletNotEnoughProduct : BOOL ;	//ERR 29 - Not enough product in the inlet
    ERR0030 : BOOL ;	//ERR 30 - not defined
    ERR0031 : BOOL ;	//ERR 31 - not defined
   END_STRUCT ;
   OutStateTarget : STRUCT 	//Command for LC, is send to LC with 'S'
    spare00 : BOOL ;
    spare01 : BOOL ;
    spare02 : BOOL ;
    spare03 : BOOL ;
    spare04 : BOOL ;
    spare05 : BOOL ;
    spare06 : BOOL ;
    spare07 : BOOL ;
    EnableEngage : BOOL ;	//Enable engage the rolls
    RestDischarge : BOOL ;	//Enable restdischarge mode (for fumigation of the bins)
    spare12 : BOOL ;
    spare13 : BOOL ;
    spare14 : BOOL ;
    spare15 : BOOL ;
    spare16 : BOOL ;
    spare17 : BOOL ;
   END_STRUCT ;
   OutComFlags : STRUCT 	//Flags for communication
    b_Done : BOOL ;	//Actual roll stand data
    S_Done : BOOL ;	//Target status
    M_Done : BOOL ;	//Target values MDDO/M
    _m_Done : BOOL ;	//Actual values MDDO/M
   END_STRUCT ;
   OutStateTargetStore : INT ;	//OutStateTarget has changed, send Cmd "S"
  END_STRUCT ;
END_VAR
VAR_TEMP
  tmpAddrOffset : DWORD ;	//store the Instance Pointer
  tmpLOGvalue : WORD ;	//LOG value
  tmpCommand : INT ;
  tmpFBNO : INT ;	//Number of the actual FB
  tmpFault : BOOL ;
  tmpWarning : BOOL ;
  tmpComActive : BOOL ;	//Put or get is in queue
  tmpLenDyn : DINT ;
  tmpAddrParFilter : DWORD ;	//Pointer to ParFilter
  tmpAddrParFilterWarning : DWORD ;	//Pointer to ParFilterWarning
  tmpAddrOutLCState : DWORD ;	//Pointer to OutLCState
  tmpAddrOutLCAlarm : DWORD ;	//Pointer to OutLCAlarm
  tmpAddrOutStateTarget : DWORD ;	//Pointer to OutLCStateTarget
  tmpComDB : INT ;
  tmpLocal : BOOL ;
  tmpHornOn : BOOL ;
END_VAR
BEGIN
NETWORK
TITLE =  Start Global
      L     35;
      T     #tmpFBNO;
      L     96;
      T     #tmpLenDyn;	//--> Len dynamic data in byte
      TAR2;
      L     DW#16#FFFFFF;
      AD;
      T     #tmpAddrOffset;	//-->Addr Para
      L     P##Par;	//[3.1]
      +D;	//[3.1]
      LAR1;
      TAR1;
      L     P#8.0;
      +D;
      T     #tmpAddrParFilter;	//-->Pointer to Par.ParFilter
      TAR1;
      L     P#12.0;
      +D;
      T     #tmpAddrParFilterWarning;	//-->Pointer to Par.ParFilterWarning
      TAR1;
      L     P#22.0;
      +D;
      T     #tmpAddrOutLCAlarm;	//-->Pointer to Par.OutLCAlarm
      TAR1;
      L     P#26.0;
      +D;
      T     #tmpAddrOutStateTarget;	//-->Pointer to Par.OutStateTarget
      L     #Par.ParComDB;
      T     #tmpComDB;
      SET;
      R     #tmpHornOn;
NETWORK
TITLE =  Call back function
//*****This functions are called by FB7 (COM) ******
      OPN   DB [#tmpComDB];
      L     0;
      L     DBW 32;	//COM.Element.CODE;
      ==I;
      JC    PC;
      L     DBB 76;	//COM.Telegram.Command;
      T     #tmpCommand;
      L     1;
      L     DBW 32;	//COM.Element.CODE;
      ==I;
      JC    Send;
      L     2;
      ==I;
      JC    Rcv;
      L     4;	//NAK
      L     DBW 32;	//COM.Element.CODE;
      ==I;
      S     #OutComFault;	//fault MDDx communication
//Handle CmdFaultReset
      A     #CmdFaultReset;
      R     #CmdFaultReset;
      S     #OutFaultResetDone;
      JU    STOR;
//Read telegram length
Send: L     #tmpCommand;
      L     'b';
      ==I;
      L     40;	//Lenght in byte
      JC    Sndx;
      L     #tmpCommand;	//[4.0]
      L     'm';	//[4.0]
      ==I;	//[4.0]
      L     36;	//Lenght in byte   //[4.0]
      JC    Sndx;	//[4.0]
      JU    SndA;
Sndx: T     DBW 86;	//COM.Telegram.LenAnswer
      JU    STOR;
SndA: NOP   0;
//Send S
      L     #tmpCommand;
      L     'S';
      <>I;
      JC    SndM;
      LAR1  #tmpAddrOutStateTarget;
      L     W [AR1,P#0.0];	// 2.0:
      T     DBD 36;	//COM.Element.InOutValue
      L     34;	//Convert Hex to 4-ASCII
      T     DBW 0;	//COM.CODE
      L     4;	//Lenght in byte
      T     DBW 78;	//COM.Telegram.Len
      CDB;	//ComDB->Instanz-DB
      UC    "GCS7_RS485Ctrl";	//Convert (CODE=DBW0)
      CDB;	//ElementDB->Instanz-DB
      JU    STOR;
//[4.0]---->
//Send M
SndM: L     #tmpCommand;
      L     'M';
      <>I;
      JC    SndZ;
//GapTopLeft    
      L     0;	//Character offset
      T     DBW 40;	//COM.Element.AddrOffset
      L     #InGapData.GapTopLeft;
      T     DBD 36;	//COM.Element.InOutValue
      L     14;	//Convert DInt to 4-ASCII
      T     DBW 0;	//COM.CODE
      CDB;	//ComDB->Instanz-DB
      UC    "GCS7_RS485Ctrl";	//Convert (CODE=DBW0)
      CDB;	//ElementDB->Instanz-DB
//GapTopRight    
      L     4;	//Character offset
      T     DBW 40;	//COM.Element.AddrOffset
      L     #InGapData.GapTopRight;
      T     DBD 36;	//COM.Element.InOutValue
      L     14;	//Convert DInt to 4-ASCII
      T     DBW 0;	//COM.CODE
      CDB;	//ComDB->Instanz-DB
      UC    "GCS7_RS485Ctrl";	//Convert (CODE=DBW0)
      CDB;	//ElementDB->Instanz-DB
//GapBottomLeft    
      L     8;	//Character offset
      T     DBW 40;	//COM.Element.AddrOffset
      L     #InGapData.GapBottomLeft;
      T     DBD 36;	//COM.Element.InOutValue
      L     14;	//Convert DInt to 4-ASCII
      T     DBW 0;	//COM.CODE
      CDB;	//ComDB->Instanz-DB
      UC    "GCS7_RS485Ctrl";	//Convert (CODE=DBW0)
      CDB;	//ElementDB->Instanz-DB
//GapBottomRight
      L     12;	//Character offset
      T     DBW 40;	//COM.Element.AddrOffset
      L     #InGapData.GapBottomRight;
      T     DBD 36;	//COM.Element.InOutValue
      L     14;	//Convert DInt to 4-ASCII
      T     DBW 0;	//COM.CODE
      CDB;	//ComDB->Instanz-DB
      UC    "GCS7_RS485Ctrl";	//Convert (CODE=DBW0)
      CDB;	//ElementDB->Instanz-DB
//Adjustment    
      L     16;	//Character offset
      T     DBW 40;	//COM.Element.AddrOffset
      L     #InGapData.GapAdjustment;
      T     DBD 36;	//COM.Element.InOutValue
      L     14;	//Convert DInt to 4-ASCII
      T     DBW 0;	//COM.CODE
      CDB;	//ComDB->Instanz-DB
      UC    "GCS7_RS485Ctrl";	//Convert (CODE=DBW0)
      CDB;	//ElementDB->Instanz-DB
      L     20;	//Lenght in byte
      T     DBW 78;	//COM.Telegram.Len
      JU    STOR;
//<--[4.0]
SndZ: JU    STOR;
//--- Get done ---------------
//Copy reveived data to element
Rcv:  R     #OutComFault;
      L     #tmpCommand;
      L     'b';
      <>I;
      JC    Rcvm;
//Feed roll speed 
      L     0;	//Character offset
      T     DBW 40;	//COM.Element.AddrOffset
      L     24;	//Convert 4-ASCII to DInt
      T     DBW 0;	//COM.CODE
      CDB;	//ComDB->Instanz-DB
      UC    "GCS7_RS485Ctrl";	//Convert (CODE=DBW0)
      CDB;	//ElementDB->Instanz-DB
      L     DBD 36;	//COM.Element.InOutValue
      T     #OutFeedRollSpeed;
//Feed roll status
      L     4;	//Character offset
      T     DBW 40;	//COM.Element.AddrOffset
      L     24;	//Convert 4-ASCII to DInt
      T     DBW 0;	//COM.CODE
      CDB;	//ComDB->Instanz-DB
      UC    "GCS7_RS485Ctrl";	//Convert (CODE=DBW0)
      CDB;	//ElementDB->Instanz-DB
      L     DBD 36;	//COM.Element.InOutValue
      T     #OutFeedRollStatus;
//Rolls up current
      L     8;	//Character offset
      T     DBW 40;	//COM.Element.AddrOffset
      L     24;	//Convert 4-ASCII to DInt
      T     DBW 0;	//COM.CODE
      CDB;	//ComDB->Instanz-DB
      UC    "GCS7_RS485Ctrl";	//Convert (CODE=DBW0)
      CDB;	//ElementDB->Instanz-DB
      L     DBD 36;	//COM.Element.InOutValue
      T     #OutRollsUpCurrent;
//Rolls low current
      L     12;	//Character offset
      T     DBW 40;	//COM.Element.AddrOffset
      L     24;	//Convert 4-ASCII to DInt
      T     DBW 0;	//COM.CODE
      CDB;	//ComDB->Instanz-DB
      UC    "GCS7_RS485Ctrl";	//Convert (CODE=DBW0)
      CDB;	//ElementDB->Instanz-DB
      L     DBD 36;	//COM.Element.InOutValue
      T     #OutRollsLowCurrent;
//Rolls up load
      L     16;	//Character offset
      T     DBW 40;	//COM.Element.AddrOffset
      L     24;	//Convert 4-ASCII to DInt
      T     DBW 0;	//COM.CODE
      CDB;	//ComDB->Instanz-DB
      UC    "GCS7_RS485Ctrl";	//Convert (CODE=DBW0)
      CDB;	//ElementDB->Instanz-DB
      L     DBD 36;	//COM.Element.InOutValue
      T     #OutRollsUpLoad;
//Rolls low load
      L     20;	//Character offset
      T     DBW 40;	//COM.Element.AddrOffset
      L     24;	//Convert 4-ASCII to DInt
      T     DBW 0;	//COM.CODE
      CDB;	//ComDB->Instanz-DB
      UC    "GCS7_RS485Ctrl";	//Convert (CODE=DBW0)
      CDB;	//ElementDB->Instanz-DB
      L     DBD 36;	//COM.Element.InOutValue
      T     #OutRollsLowLoad;
//Grind gap status
      L     24;	//Character offset
      T     DBW 40;	//COM.Element.AddrOffset
      L     24;	//Convert 4-ASCII to DInt
      T     DBW 0;	//COM.CODE
      CDB;	//ComDB->Instanz-DB
      UC    "GCS7_RS485Ctrl";	//Convert (CODE=DBW0)
      CDB;	//ElementDB->Instanz-DB
      L     DBD 36;	//COM.Element.InOutValue
      T     #OutGrindGapStatus;
//Alarm number
      L     28;	//Character offset
      T     DBW 40;	//COM.Element.AddrOffset
      L     24;	//Convert 4-ASCII to DInt
      T     DBW 0;	//COM.CODE
      CDB;	//ComDB->Instanz-DB
      UC    "GCS7_RS485Ctrl";	//Convert (CODE=DBW0)
      CDB;	//ElementDB->Instanz-DB
      L     DBD 36;	//COM.Element.InOutValue
      T     #OutAlarmNr;
//Reserve
      L     32;	//Character offset
      T     DBW 40;	//COM.Element.AddrOffset
      L     24;	//Convert 4-ASCII to DInt
      T     DBW 0;	//COM.CODE
      CDB;	//ComDB->Instanz-DB
      UC    "GCS7_RS485Ctrl";	//Convert (CODE=DBW0)
      CDB;	//ElementDB->Instanz-DB
      L     DBD 36;	//COM.Element.InOutValue
      T     #spare2200;
//LC status
      L     36;	//Character offset
      T     DBW 40;	//COM.Element.AddrOffset
      L     44;	//Convert 4-ASCII to Hex
      T     DBW 0;	//COM.CODE
      CDB;	//ComDB->Instanz-DB
      UC    "GCS7_RS485Ctrl";	//Convert (CODE=DBW0)
      CDB;	//ElementDB->Instanz-DB
      L     #tmpAddrOffset;	//-->Addr Para
      L     P##OutLCState;
      +D;
      LAR1;
      L     DBD 36;	//COM.Element.InOutValue
      T     W [AR1,P#0.0];	//#OutLCState
//Handle CmdFaultReset
      A     #CmdFaultReset;
      R     #CmdFaultReset;
      S     #OutFaultResetDone;
      JU    STOR;
//[4.0]-->
//Command 'm'
Rcvm: R     #OutComFault;
      L     #tmpCommand;
      L     'm';
      <>I;
      JC    RcvM;
//GapTopLeftNom
      L     0;	//Character offset
      T     DBW 40;	//COM.Element.AddrOffset
      L     24;	//Convert 4-ASCII to DInt
      T     DBW 0;	//COM.CODE
      CDB;	//ComDB->Instanz-DB
      UC    "GCS7_RS485Ctrl";	//Convert (CODE=DBW0)
      CDB;	//ElementDB->Instanz-DB
      L     DBD 36;	//COM.Element.InOutValue
      T     #OutGapData.GapTopLeftNom;
//GapTopRightNom
      L     4;	//Character offset
      T     DBW 40;	//COM.Element.AddrOffset
      L     24;	//Convert 4-ASCII to DInt
      T     DBW 0;	//COM.CODE
      CDB;	//ComDB->Instanz-DB
      UC    "GCS7_RS485Ctrl";	//Convert (CODE=DBW0)
      CDB;	//ElementDB->Instanz-DB
      L     DBD 36;	//COM.Element.InOutValue
      T     #OutGapData.GapTopRightNom;
//GapBottomLeftNom
      L     8;	//Character offset
      T     DBW 40;	//COM.Element.AddrOffset
      L     24;	//Convert 4-ASCII to DInt
      T     DBW 0;	//COM.CODE
      CDB;	//ComDB->Instanz-DB
      UC    "GCS7_RS485Ctrl";	//Convert (CODE=DBW0)
      CDB;	//ElementDB->Instanz-DB
      L     DBD 36;	//COM.Element.InOutValue
      T     #OutGapData.GapBottomLeftNom;
//GapBottomRightNom
      L     12;	//Character offset
      T     DBW 40;	//COM.Element.AddrOffset
      L     24;	//Convert 4-ASCII to DInt
      T     DBW 0;	//COM.CODE
      CDB;	//ComDB->Instanz-DB
      UC    "GCS7_RS485Ctrl";	//Convert (CODE=DBW0)
      CDB;	//ElementDB->Instanz-DB
      L     DBD 36;	//COM.Element.InOutValue
      T     #OutGapData.GapBottomRightNom;
//GapTopLeftAc
      L     16;	//Character offset
      T     DBW 40;	//COM.Element.AddrOffset
      L     24;	//Convert 4-ASCII to DInt
      T     DBW 0;	//COM.CODE
      CDB;	//ComDB->Instanz-DB
      UC    "GCS7_RS485Ctrl";	//Convert (CODE=DBW0)
      CDB;	//ElementDB->Instanz-DB
      L     DBD 36;	//COM.Element.InOutValue
      T     #OutGapData.GapTopLeftAc;
//GapTopRightAc
      L     20;	//Character offset
      T     DBW 40;	//COM.Element.AddrOffset
      L     24;	//Convert 4-ASCII to DInt
      T     DBW 0;	//COM.CODE
      CDB;	//ComDB->Instanz-DB
      UC    "GCS7_RS485Ctrl";	//Convert (CODE=DBW0)
      CDB;	//ElementDB->Instanz-DB
      L     DBD 36;	//COM.Element.InOutValue
      T     #OutGapData.GapTopRightAc;
//GapBottomLeftAc
      L     24;	//Character offset
      T     DBW 40;	//COM.Element.AddrOffset
      L     24;	//Convert 4-ASCII to DInt
      T     DBW 0;	//COM.CODE
      CDB;	//ComDB->Instanz-DB
      UC    "GCS7_RS485Ctrl";	//Convert (CODE=DBW0)
      CDB;	//ElementDB->Instanz-DB
      L     DBD 36;	//COM.Element.InOutValue
      T     #OutGapData.GapBottomLeftAc;
//GapBottomRightAc
      L     28;	//Character offset
      T     DBW 40;	//COM.Element.AddrOffset
      L     24;	//Convert 4-ASCII to DInt
      T     DBW 0;	//COM.CODE
      CDB;	//ComDB->Instanz-DB
      UC    "GCS7_RS485Ctrl";	//Convert (CODE=DBW0)
      CDB;	//ElementDB->Instanz-DB
      L     DBD 36;	//COM.Element.InOutValue
      T     #OutGapData.GapBottomRightAc;
//Adjustment
      L     32;	//Character offset
      T     DBW 40;	//COM.Element.AddrOffset
      L     24;	//Convert 4-ASCII to DInt
      T     DBW 0;	//COM.CODE
      CDB;	//ComDB->Instanz-DB
      UC    "GCS7_RS485Ctrl";	//Convert (CODE=DBW0)
      CDB;	//ElementDB->Instanz-DB
      L     DBD 36;	//COM.Element.InOutValue
      T     #OutGapData.GapAdjustment;
      JU    STOR;
//<--[4.0]
//--- Put done ---------------
RcvM: L     #tmpCommand;	//[4.0]
      L     'M';	//[4.0]
      <>I;	//[4.0]
      JC    RcvS;	//[4.0]
      R     #CmdNewValue;	//[4.0]
      JU    STOR;	//[4.0]
RcvS: L     #tmpCommand;
      L     'S';
      <>I;
      JC    RcvX;
RcvX: JU    STOR;
NETWORK
TITLE = PC Control
//=== Test Object number =====================
PC:   L     "SYS_DirectCtrlDB".PC.ObjectNo;	//PCControl.ObjectNo
      L     #Par.ParObjectNo;	//Input ObjectNo
      <>I;
      JC    Ctrl;
//=== Test OType      ========================
      L     1035;	//Input object type
      L     "SYS_DirectCtrlDB".PC.ObjectType;	//PCControl.ObjectType
      <>I;
      JC    Ctrl;
//=== Test Handshake =========================
      A     "SYS_DirectCtrlDB".PC.Hsk.FExamine;	//Handshake.FExamine
      JC    pExa;
      A     "SYS_DirectCtrlDB".PC.Hsk.FDefineCmd;	//Handshake.FDefineCmd
      JC    pCmd;
      A     "SYS_DirectCtrlDB".PC.Hsk.FDefinePara;	//Handshake.FDefinePara
      JC    pPar;
pIni: L     2;	//FcInit
      UC    "SYS_DirectCtrl";
      JU    Ctrl;
//Write parameter 
pPar: NOP   0;
//Write new commands from PC to Interface of group 
pCmd: A     "SYS_DirectCtrlDB".PC.Cmd1[11];	//Cmd1[11] =CmdFaultReset
      S     #CmdFaultReset;
      JU    pIni;
pExa: TAR2;	//Address dynamic datas
      T     "SYS_DirectCtrlDB".GC.InDynAddr;	//-->PCControl.GC.InDynAddr
      L     #tmpLenDyn;	//Length dynamic datas
      T     "SYS_DirectCtrlDB".GC.InDynLen;	//-->PCControl.GC.InDynLen
      L     0;
      T     "SYS_DirectCtrlDB".GC.InParaAddr;	//-->PCControl.GC.InParaAddr
      T     "SYS_DirectCtrlDB".GC.InParaLen;	//-->PCControl.GC.InParaLen
      L     1;	//Code FcExamine
      UC    "SYS_DirectCtrl";
      L     11;	//Revision
      T     "SYS_DirectCtrlDB".GC.Revision;
NETWORK
TITLE =  Read LC data
Ctrl: OPN   DB [#tmpComDB];
      L     #Par.ParLCIdx;
      T     DBW 34;	//COM.Element.Index;
      L     1;	//Read LC data
      T     DBW 0;	//COM.CODE;
      CDB;
      UC    "GCS7_RS485Ctrl";
      CDB;
      L     #tmpFBNO;
      T     DBW 52;	//COM.LC0.FBNO;   
      L     DINO;
      T     DBW 54;	//COM.LC0.DINO;
      TAR2  DBD 56;	//COM.LC0.AddrDyn;        
      L     #tmpAddrOffset;
      T     DBD 60;	//COM.LC0.AddrPara;       
      L     #Par.ParLCAddr;
      T     DBD 64;	//COM.Telegram.LCAddr;
NETWORK
TITLE =  All State Init
//===Clear tmp Variable
//===Global Group Orders===
      A     #InLocal;
      O     #InDPFault;
      O     #InHWStop;
      =     #tmpLocal;
//---FaultReset is on---
      A     "GCS7_Gr_OutFaultReset";	//Gr.OutFaultReset
      S     #CmdFaultReset;
//--- tmpFault   
      L     #OutAlarmNr;	//Calculate OutLCAlarm out of the AlarmNumber
      L     1;
      SLD;
      SRD   1;	//Clear Alarm Bit 0
      SLD   1;
      CAD;	//Replace akku to correct bit order
      LAR1  #tmpAddrOutLCAlarm;
      T     D [AR1,P#0.0];	//#OutLCAlarm
      LAR1  #tmpAddrParFilter;
      L     D [AR1,P#0.0];	//#Par.ParFilter;
      INVD;	//Invers filter mask
      AD;
      L     0;
      <>D;
      O     #OutComFault;	//---Communication fault
      =     #tmpFault;
//      TAK                             // 2.1:
      LAR1  #tmpAddrOutLCAlarm;	// 2.1:
      L     D [AR1,P#0.0];	// 2.1: #OutLCAlarm
      LAR1  #tmpAddrParFilterWarning;
      L     D [AR1,P#0.0];	//#Par.ParFilterWarning;
      AD;
      L     0;
      <>D;
      AN    #OutComFault;
      O;
      A     #OutComFault;	//Warning mode: for OutComFault
      A     #Par.ParWarning;	//if ParWarning is set
      =     #tmpWarning;	//additional information (tmpFault is also set)
      A     DBX 50.0;	//COM.LC0.CmdPut
      O     DBX 50.1;	//COM.LC0.CmdGet
      =     #tmpComActive;
//---LC State target commands
      A     #InEnableEngage;
      =     #Par.OutStateTarget.EnableEngage;
      A     #InRestdischarge;
      =     #Par.OutStateTarget.RestDischarge;
NETWORK
TITLE = Communication start
      A     #tmpComActive;
      JC    STAT;
      L     #Par.OutStateTargetStore;	// 2.0:---State target has changed?
      LAR1  #tmpAddrOutStateTarget;	// 2.0:   -> Send command S
      L     W [AR1,P#0.0];	// 2.0:
      <>I;	// 2.0:
      AN    #Par.OutComFlags.S_Done;
      JC    CmdS;
      AN    #Par.OutComFlags.b_Done;
      JC    Cmdb;
      AN    #Par.OutComFlags.M_Done;	//[4.0]
      A     #CmdNewValue;	//[4.0]
      A     #Par.ParNoMDEF;	//[4.0]
      JC    CmdM;	//[4.0]
      AN    #Par.OutComFlags._m_Done;	//[4.0]
      A     #Par.ParNoMDEF;	//[4.0]
      JC    Cmdm;	//[4.0]
      R     #Par.OutComFlags.b_Done;	//[4.0]
      R     #Par.OutComFlags.S_Done;
      R     #Par.OutComFlags.M_Done;	//[4.0]
      R     #Par.OutComFlags._m_Done;	//[4.0]
      JU    OUT;
Cmdb: S     #Par.OutComFlags.b_Done;
      L     'b';
      JU    GET;
Cmdm: S     #Par.OutComFlags._m_Done;	//[4.0]
      L     'm';	//[4.0]
      JU    GET;	//[4.0]
CmdS: T     #Par.OutStateTargetStore;	// 2.0:---Store state target
      S     #Par.OutComFlags.S_Done;
      L     'S';
      JU    PUT;
CmdM: S     #Par.OutComFlags.M_Done;	//[4.0]
      L     'M';	//[4.0]
      JU    PUT;	//[4.0]
PUT:  SET;
      S     DBX 50.0;	//COM.LC0.CmdPut;
      JU    ALL1;
GET:  SET;
      S     DBX 50.1;	//COM.LC0.CmdGet;
ALL1: S     #tmpComActive;
      T     DBB 51;	//COM.LC0.Command;
      JU    OUT;
NETWORK
TITLE = States
//===State machine===
STAT: A     #StOk;
      JC    S2;
      A     #StFault;
      JC    S4;
      A     #StWarning;
      JC    S5;
      S     #StOk;	//Init
NETWORK
TITLE =  StOk
xS2:  S     #StOk;
      R     #StWarning;
      R     #StFault;
      R     #CmdFaultReset;
      R     #OutFaultResetDone;
      L     B#(3, 9);	//Message Operator ('fault cancelled' )
      JU    LOG;
S2:   A     #tmpWarning;	//---Condition to set Horn
      O     #tmpFault;	// 2.0:
      AN    #tmpLocal;	// 2.0:
      S     #tmpHornOn;
      A     #tmpWarning;	// 2.0:---Condition for StFault/StWarning
      O     #tmpFault;	// 2.0:
      JC    xS45;	//StXxx -> StFault/StWarning transition
      JU    OUT;
NETWORK
TITLE =  StFault
S4:   AN    #tmpFault;	//---Condition for StOk
      A     #CmdFaultReset;
      JC    xS2;
      A     #InLocal;	//---Condition for StWarning
      O     #tmpWarning;
      JC    xS45;
      A     #OutFaultResetDone;	//reLOG fault
      JC    xS45;
      JU    OUT;
NETWORK
TITLE =  StWarning
//Automatic fault reset
S5:   AN    #tmpFault;	//---Condition for StOk
      AN    #tmpWarning;	// 2.1:
      A     #InLocal;	// 2.1:
      O;	// 2.1:
      AN    #tmpWarning;	// 2.1:
      AN    #tmpFault;	// 2.1:
      AN    #InLocal;	// 2.1:
      A     #CmdFaultReset;	// 2.1:
      JC    xS2;
      AN    #tmpLocal;	//---Condition for StFault
      AN    #tmpWarning;
      A     #tmpFault;	// 2.1:
      S     #tmpHornOn;
      JC    xS45;	//StXxx -> StFault transition flag
      AN    #InLocal;	//2.1: reLOG warning
      A     #OutFaultResetDone;	// 2.1:
      JC    xS45;	// 2.1:
      A     #OutFaultResetDone;	//---Fault reset
      S     #CmdFaultReset;
      R     #OutFaultResetDone;
      JU    OUT;
NETWORK
TITLE = LOG
xS45: R     #StOk;
      R     #OutFaultResetDone;	//---Fault reset
//---Horn On-----------------------------
      AN    #tmpHornOn;
      JC    S4J2;
      S     "GCS7_Gr_InFaultFlag";	// Gr.InFaultFlag
      CALL  "SYS_Horn_Code" (
           FcCode                   := 1,
           ParObjectType            := 1035,
           ParObjectNo              := #Par.ParObjectNo,
           ParHornCode              := #Par.ParHornCode);
//---Message------------------------------
S4J2: A     #tmpLocal;	//----Condition for StWarning
      O     #tmpWarning;
      S     #StWarning;
      R     #StFault;
      A     #tmpLocal;	// 2.1:---InLocal=1 -> no LOG message
      JC    OUT;
      A     #tmpFault;	// 2.1:
      AN    #tmpWarning;	// 2.1:
      S     #StFault;
      R     #StWarning;
      L     B#(1, 10);
      A     #OutComFault;
      JC    LOG;
      L     B#(1, 1);
      A     #Par.OutLCAlarm.CheckSumFault;
      JC    LOG;
      L     B#(1, 2);
      A     #Par.OutLCAlarm.RAMTestFault;
      JC    LOG;
      L     B#(1, 3);
      A     #Par.OutLCAlarm.OperationFault;
      JC    LOG;
      L     B#(1, 4);
      A     #Par.OutLCAlarm.WatchDog;
      JC    LOG;
      L     B#(1, 5);
      A     #Par.OutLCAlarm.MemoryLost;
      JC    LOG;
      L     B#(1, 6);
      A     #Par.OutLCAlarm.GrindGapPrint;
      JC    LOG;
      L     B#(1, 7);	// 2.0:
      A     #Par.OutLCAlarm.ERR0007;
      JC    LOG;
      L     B#(1, 8);	// 2.0:
      A     #Par.OutLCAlarm.ERR0008;
      JC    LOG;
      L     B#(1, 11);
      A     #Par.OutLCAlarm.GrindRollsDryRun;
      JC    LOG;
      L     B#(1, 12);	// 2.0:
      A     #Par.OutLCAlarm.ERR0012;
      JC    LOG;
      L     B#(1, 13);
      A     #Par.OutLCAlarm.FeedRollsStandstill;
      JC    LOG;
      L     B#(1, 14);
      A     #Par.OutLCAlarm.GrindRollsStandstill;
      JC    LOG;
      L     B#(1, 15);
      A     #Par.OutLCAlarm.GrindRollsLowStandstill;
      JC    LOG;
      L     B#(1, 16);
      A     #Par.OutLCAlarm.MotorOverload;
      JC    LOG;
      L     B#(1, 17);
      A     #Par.OutLCAlarm.MotorLowOverload;
      JC    LOG;
      L     B#(1, 18);
      A     #Par.OutLCAlarm.GrindGapFault;
      JC    LOG;
      L     B#(1, 19);
      A     #Par.OutLCAlarm.GrindGapLowFault;
      JC    LOG;
      L     B#(1, 20);
      A     #Par.OutLCAlarm.ProdRegistrationFault;
      JC    LOG;
      L     B#(1, 21);
      A     #Par.OutLCAlarm.GrindGapNoIncr;
      JC    LOG;
      L     B#(1, 22);
      A     #Par.OutLCAlarm.GrindGapLowNoIncr;
      JC    LOG;
      L     B#(1, 23);
      A     #Par.OutLCAlarm.HLInlet;
      JC    LOG;
      L     B#(1, 24);
      A     #Par.OutLCAlarm.HLOutlet;
      JC    LOG;
      L     B#(1, 25);
      A     #Par.OutLCAlarm.HLBackUpLeft;
      JC    LOG;
      L     B#(1, 26);
      A     #Par.OutLCAlarm.HLBackUpRight;
      JC    LOG;
      L     B#(1, 27);
      A     #Par.OutLCAlarm.EmergencyStop;
      JC    LOG;
      L     B#(1, 28);	// 2.0:
      A     #Par.OutLCAlarm.InletProductFullRpnmax;
      JC    LOG;
      L     B#(1, 29);	// 2.0:
      A     #Par.OutLCAlarm.InletNotEnoughProduct;
      JC    LOG;
      L     B#(1, 30);	// 2.0:
      A     #Par.OutLCAlarm.ERR0030;
      JC    LOG;
      L     B#(1, 31);	// 2.0:
      A     #Par.OutLCAlarm.ERR0031;
      JC    LOG;
      L     B#(1, 10);	//COM communication
      JU    LOG;
LOG:  A     #Par.ParLogOff;	//---Set LOG Message
      JC    SAVE;
      T     #tmpLOGvalue;
      L     W#16#FF;
      AW;
      T     #OutAlarmNrLog;
      CALL  "GCS7_LogConvert" (
           ObjectNo                 := #Par.ParObjectNo,
           MsgType                  := #Par.ParMsgType,
           ClassMsgTxt              := #tmpLOGvalue,
           OType                    := 1035);	//LOG Message Converter / Entry / Contains Class and TextNo
NETWORK
TITLE = Global End
OUT:  NOP   0;
SAVE: SET;	//---Clear all commands
//--Output for group 
      A     #InDPFault;
      AN    #InLocal;
      S     "GCS7_Gr_InDPFault";
      A     #InHWStop;
      AN    #InLocal;
      S     "GCS7_Gr_InHWStop";
NETWORK
TITLE = State Code
      L     3;	//Code: ok
      A     #StOk;
      JC    STC;
//--Warning ---
      AN    #StWarning;
      JC    STC2;
      L     45;	//Code:StWarning.HWStop
      A     #InHWStop;
      JC    STC;
      L     55;	//Code: StWarning.DPFault
      A     #InDPFault;
      JC    STC;
      L     5;	//Code: StWarning
      JU    STC;
//===============
STC2: L     32;	//Code: fault
STC:  L     #StCode;	//Old state code
      TAK;
      T     #StCode;	//Save state code
      <>I;
      L     3;	//Load code for CBit methode
      CC    "SYS_CBitCtrl";
NETWORK
TITLE =  Store LC data
      L     #Par.ParLCIdx;
      T     DBW 34;	//COM.Element.Index; 
      L     2;	//Store LC data
      T     DBW 0;	//COM.CODE;
      CDB;
      UC    "GCS7_RS485Ctrl";
      CDB;
STOR: NOP   0;
END_FUNCTION_BLOCK

